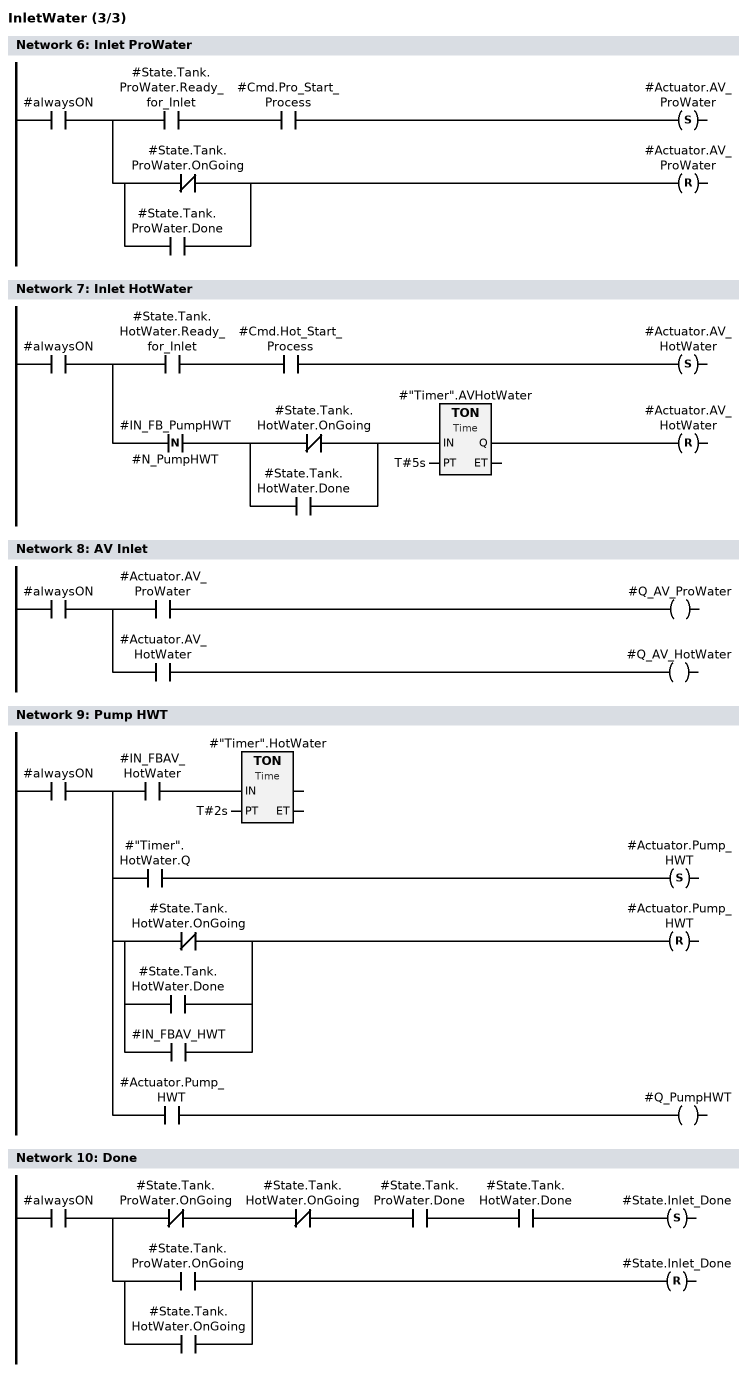
   RUNG wire#powerrail
      Contact( #alwaysON )
      wire#w1
      Contact( #State.Tank.ProWater.Ready_for_Inlet )
      Contact( #Cmd.Pro_Start_Process )
      S_Coil( #Actuator.AV_ProWater )
   END_RUNG
   RUNG wire#w1
      I_Contact( #State.Tank.ProWater.OnGoing )
      wire#w2
      R_Coil( #Actuator.AV_ProWater )
   END_RUNG
   RUNG wire#w1
      Contact( #State.Tank.ProWater.Done )
   END_RUNG wire#w2
   // the same network as SCL:
   IF #alwaysON AND #State.Tank.ProWater.Ready_for_Inlet AND #Cmd.Pro_Start_Process THEN
       #Actuator.AV_ProWater := TRUE;
   END_IF;
   IF #alwaysON AND (NOT #State.Tank.ProWater.OnGoing OR #State.Tank.ProWater.Done) THEN
       #Actuator.AV_ProWater := FALSE;
   END_IF;
END_REGION

REGION Network 7: Inlet HotWater
   RUNG wire#powerrail
      Contact( #alwaysON )
      wire#w1
      Contact( #State.Tank.HotWater.Ready_for_Inlet )
      Contact( #Cmd.Hot_Start_Process )
      S_Coil( #Actuator.AV_HotWater )
   END_RUNG
   RUNG wire#w1
      N_Contact(operand := #IN_FB_PumpHWT, bit := #N_PumpHWT)
      wire#w2
      I_Contact( #State.Tank.HotWater.OnGoing )
      wire#w3
      { S7_Templates := "time_type := Time" } #"Timer".AVHotWater.TON(pt := T#5s, et =>)
      R_Coil( #Actuator.AV_HotWater )
   END_RUNG
   RUNG wire#w2
      Contact( #State.Tank.HotWater.Done )
   END_RUNG wire#w3
   // the same network as SCL:
   IF #alwaysON AND #State.Tank.HotWater.Ready_for_Inlet AND #Cmd.Hot_Start_Process THEN
       #Actuator.AV_HotWater := TRUE;
   END_IF;
   #_w1 := #alwaysON AND NOT #IN_FB_PumpHWT AND #N_PumpHWT;   // falling edge of #IN_FB_PumpHWT
   #N_PumpHWT := #IN_FB_PumpHWT;
   #"Timer".AVHotWater.TON(IN := #_w1 AND (NOT #State.Tank.HotWater.OnGoing OR #State.Tank.HotWater.Done),
                           PT := T#5s);
   IF #"Timer".AVHotWater.Q THEN #Actuator.AV_HotWater := FALSE; END_IF;
END_REGION

REGION Network 8: AV Inlet
   RUNG wire#powerrail
      Contact( #alwaysON )
      wire#w1
      Contact( #Actuator.AV_ProWater )
      Coil( #Q_AV_ProWater )
   END_RUNG
   RUNG wire#w1
      Contact( #Actuator.AV_HotWater )
      Coil( #Q_AV_HotWater )
   END_RUNG
   // the same network as SCL:
   #Q_AV_ProWater := #alwaysON AND #Actuator.AV_ProWater;
   #Q_AV_HotWater := #alwaysON AND #Actuator.AV_HotWater;
END_REGION

REGION Network 9: Pump HWT
   RUNG wire#powerrail
      Contact( #alwaysON )
      wire#w1
      Contact( #IN_FBAV_HotWater )
      { S7_Templates := "time_type := Time" } #"Timer".HotWater.TON(pt := T#2s, et =>)
   END_RUNG
   RUNG wire#w1
      Contact( #"Timer".HotWater.Q )
      S_Coil( #Actuator.Pump_HWT )
   END_RUNG
   RUNG wire#w1
      I_Contact( #State.Tank.HotWater.OnGoing )
      wire#w2
      R_Coil( #Actuator.Pump_HWT )
   END_RUNG
   RUNG wire#w1
      Contact( #State.Tank.HotWater.Done )
   END_RUNG wire#w2
   RUNG wire#w1
      Contact( #IN_FBAV_HWT )
   END_RUNG wire#w2
   RUNG wire#w1
      Contact( #Actuator.Pump_HWT )
      Coil( #Q_PumpHWT )
   END_RUNG
   // the same network as SCL:
   #"Timer".HotWater.TON(IN := #alwaysON AND #IN_FBAV_HotWater, PT := T#2s);
   IF #alwaysON AND #"Timer".HotWater.Q THEN #Actuator.Pump_HWT := TRUE; END_IF;
   IF #alwaysON AND (NOT #State.Tank.HotWater.OnGoing OR #State.Tank.HotWater.Done OR #IN_FBAV_HWT) THEN
       #Actuator.Pump_HWT := FALSE;
   END_IF;
   #Q_PumpHWT := #alwaysON AND #Actuator.Pump_HWT;
END_REGION

REGION Network 10: Done
   RUNG wire#powerrail
      Contact( #alwaysON )
      wire#w1
      I_Contact( #State.Tank.ProWater.OnGoing )
      I_Contact( #State.Tank.HotWater.OnGoing )
      Contact( #State.Tank.ProWater.Done )
      Contact( #State.Tank.HotWater.Done )
      S_Coil( #State.Inlet_Done )
   END_RUNG
   RUNG wire#w1
      Contact( #State.Tank.ProWater.OnGoing )
      wire#w2
      R_Coil( #State.Inlet_Done )
   END_RUNG
   RUNG wire#w1
      Contact( #State.Tank.HotWater.OnGoing )
   END_RUNG wire#w2
   // the same network as SCL:
   IF #alwaysON AND NOT #State.Tank.ProWater.OnGoing AND NOT #State.Tank.HotWater.OnGoing AND #State.Tank.ProWater.Done AND #State.Tank.HotWater.Done THEN
       #State.Inlet_Done := TRUE;
   END_IF;
   IF #alwaysON AND (#State.Tank.ProWater.OnGoing OR #State.Tank.HotWater.OnGoing) THEN
       #State.Inlet_Done := FALSE;
   END_IF;
END_REGION
END_FUNCTION_BLOCK

FUNCTION_BLOCK "Storage Tank"   // FB7, LAD
{ S7_Optimized_Access := 'TRUE' }
VERSION : 0.1
// stored: AutoNumber true, IsIECCheckEnabled false, IsRetainMemResEnabled false, MemoryReserve 100, SetENOAutomatically false, UDAEnableTagReadback false
   VAR_INPUT
      Lock : Bool;
      Reset : Bool;
   END_VAR
   VAR_OUTPUT
      AV_Inlet : Bool;
   END_VAR
   VAR_IN_OUT
      Tank_Level : Real;
   END_VAR
   VAR
      Parameter : Struct
         Level_High : Real := 100.0;
         Level_Med : Real := 50.0;
         Level_Low : Real;
      END_STRUCT;
      State : Struct
         Tank_HL : Bool;
         Tank_ML : Bool;
         Tank_LL : Bool;
      END_STRUCT;
      Actuator : Struct
         AV_Inlet : Bool;
      END_STRUCT;
      AlwaysOn : Bool;
      Stat_Ready_for_Transfer : Bool;
      Ready_for_Transfer : Bool;
   END_VAR
BEGIN

REGION Network 1: Always On
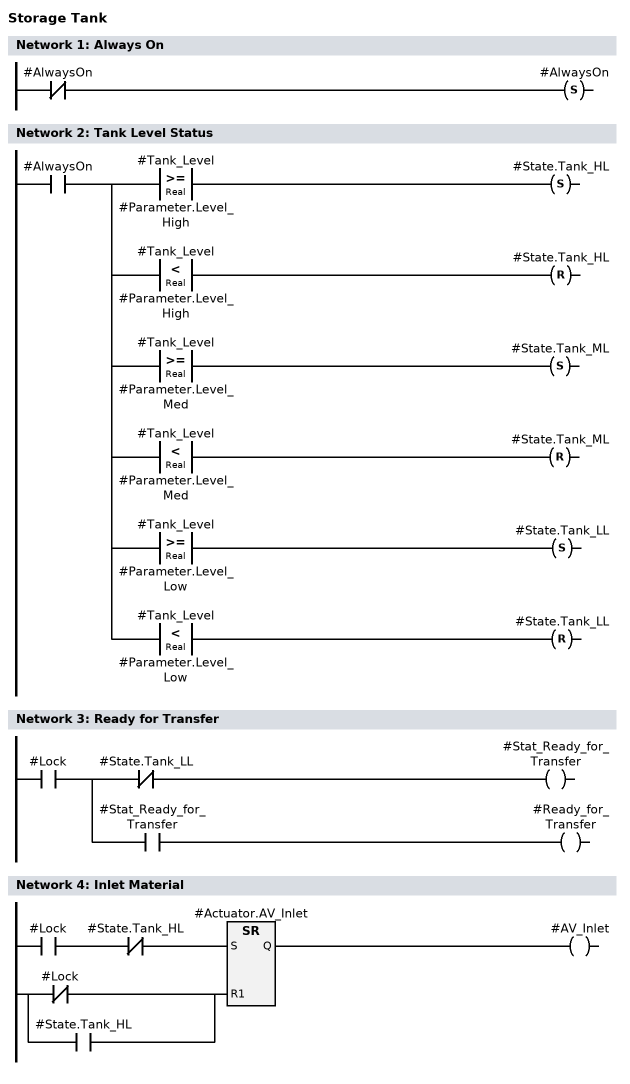
   RUNG wire#powerrail
      I_Contact( #AlwaysOn )
      S_Coil( #AlwaysOn )
   END_RUNG
   // the same network as SCL:
   IF NOT #AlwaysOn THEN #AlwaysOn := TRUE; END_IF;
END_REGION

REGION Network 2: Tank Level Status
   RUNG wire#powerrail
      Contact( #AlwaysOn )
      wire#w1
      { S7_Templates := "SrcType := Real" } GE_Contact(in1 := #Tank_Level, in2 := #Parameter.Level_High)
      S_Coil( #State.Tank_HL )
   END_RUNG
   RUNG wire#w1
      { S7_Templates := "SrcType := Real" } LT_Contact(in1 := #Tank_Level, in2 := #Parameter.Level_High)
      R_Coil( #State.Tank_HL )
   END_RUNG
   RUNG wire#w1
      { S7_Templates := "SrcType := Real" } GE_Contact(in1 := #Tank_Level, in2 := #Parameter.Level_Med)
      S_Coil( #State.Tank_ML )
   END_RUNG
   RUNG wire#w1
      { S7_Templates := "SrcType := Real" } LT_Contact(in1 := #Tank_Level, in2 := #Parameter.Level_Med)
      R_Coil( #State.Tank_ML )
   END_RUNG
   RUNG wire#w1
      { S7_Templates := "SrcType := Real" } GE_Contact(in1 := #Tank_Level, in2 := #Parameter.Level_Low)
      S_Coil( #State.Tank_LL )
   END_RUNG
   RUNG wire#w1
      { S7_Templates := "SrcType := Real" } LT_Contact(in1 := #Tank_Level, in2 := #Parameter.Level_Low)
      R_Coil( #State.Tank_LL )
   END_RUNG
   // the same network as SCL:
   IF #AlwaysOn AND (#Tank_Level >= #Parameter.Level_High) THEN #State.Tank_HL := TRUE; END_IF;
   IF #AlwaysOn AND (#Tank_Level < #Parameter.Level_High) THEN #State.Tank_HL := FALSE; END_IF;
   IF #AlwaysOn AND (#Tank_Level >= #Parameter.Level_Med) THEN #State.Tank_ML := TRUE; END_IF;
   IF #AlwaysOn AND (#Tank_Level < #Parameter.Level_Med) THEN #State.Tank_ML := FALSE; END_IF;
   IF #AlwaysOn AND (#Tank_Level >= #Parameter.Level_Low) THEN #State.Tank_LL := TRUE; END_IF;
   IF #AlwaysOn AND (#Tank_Level < #Parameter.Level_Low) THEN #State.Tank_LL := FALSE; END_IF;
END_REGION

REGION Network 3: Ready for Transfer
   RUNG wire#powerrail
      Contact( #Lock )
      wire#w1
      I_Contact( #State.Tank_LL )
      Coil( #Stat_Ready_for_Transfer )
   END_RUNG
   RUNG wire#w1
      Contact( #Stat_Ready_for_Transfer )
      Coil( #Ready_for_Transfer )
   END_RUNG
   // the same network as SCL:
   #Stat_Ready_for_Transfer := #Lock AND NOT #State.Tank_LL;
   #Ready_for_Transfer := #Lock AND #Stat_Ready_for_Transfer;
END_REGION

REGION Network 4: Inlet Material
   RUNG wire#powerrail
      Contact( #Lock )
      I_Contact( #State.Tank_HL )
      S_SR(operand := #Actuator.AV_Inlet, r1 := wire#w1)
      Coil( #AV_Inlet )
   END_RUNG
   RUNG wire#powerrail
      I_Contact( #Lock )
   END_RUNG wire#w1
   RUNG wire#powerrail
      Contact( #State.Tank_HL )
   END_RUNG wire#w1
   // the same network as SCL:
   IF #Lock AND NOT #State.Tank_HL THEN
       #Actuator.AV_Inlet := TRUE;   // SR flip-flop
   END_IF;
   IF NOT #Lock OR #State.Tank_HL THEN #Actuator.AV_Inlet := FALSE; END_IF;
   #AV_Inlet := #Actuator.AV_Inlet;
END_REGION
END_FUNCTION_BLOCK

FUNCTION "IO Blending" : Void   // FC3, LAD
{ S7_Optimized_Access := 'TRUE' }
VERSION : 0.1
// stored: AutoNumber true, IsIECCheckEnabled false, SetENOAutomatically false, UDAEnableTagReadback false
BEGIN
END_FUNCTION

FUNCTION_BLOCK "IO_Valve_Blending"   // FB2, LAD
{ S7_Optimized_Access := 'FALSE' }
VERSION : 0.1
// stored: AutoNumber true, IsIECCheckEnabled false, SetENOAutomatically false, UDAEnableTagReadback false
   VAR_INPUT
      lock : Bool;
      Init : Bool;
      Reset : Bool;
   END_VAR
   VAR
      "AV-20.01" { S7_SetPoint := 'True'} : "Valve";   // AUTO BUTTERFLY VALVE OUTLET PRODUCT BLENDING TANK T-20.00
      "AV-20.02" { S7_SetPoint := 'True'} : "Valve";   // AUTO BUTTERGLY VALVE INLET CIP SUPPLY LINE BLENDING TANK T-20.00
      "AV-20.03" { S7_SetPoint := 'True'} : "Valve";   // AUTO BUTTERFLY VALVE OUTLET PRODUCT FROM BLENDING T-20.00 TO TRANSFER PUMP P-21.01
      "AV-20.04" { S7_SetPoint := 'True'} : "Valve";   // AUTO BUTTERFLY VALVE CIP RETURN FROM BLENDING TANK T-20.00
      "AV-20.05" { S7_SetPoint := 'True'} : "Valve";   // AUTO BUTTERFLY VALVE INLET FRESH CHILI FROM T-06.00 TO BLENDING TANK T-20.00
      "AV-20.06" { S7_SetPoint := 'True'} : "Valve";   // AUTO BUTTERFLY VALVE INLET FRESH CHILI FROM T-07.00 TO BLENDING TANK T-20.00
      "AV-20.07" { S7_SetPoint := 'True'} : "Valve";   // AUTO BUTTERFLY VALVE INLET FRESH CHILI FROM T-08.00 TO BLENDING TANK T-20.00
      "AV-20.08" { S7_SetPoint := 'True'} : "Valve";   // AUTO BUTTERFLY VALVE INLET GARLIC FROM T-09.00 TO BLENDING TANK T-20.00
      "AV-20.09" { S7_SetPoint := 'True'} : "Valve";   // AUTO BUTTERFLY VALVE INLET CHILI AWETAN FROM T-02.00 TO BLENDING TANK T-20.00
      "AV-20.10" { S7_SetPoint := 'True'} : "Valve";   // AUTO BUTTERFLY VALVE INLET CHILI AWETAN FROM T-03.00 TO BLENDING TANK T-20.00
      "AV-20.11" { S7_SetPoint := 'True'} : "Valve";   // AUTO BUTTERFLY VALVE INLET CHILI AWETAN FROM T-04.00 TO BLENDING TANK T-20.00
      "AV-20.12" { S7_SetPoint := 'True'} : "Valve";   // AUTO BUTTERFLY VALVE INLET TOMATO FROM T-05.00 TO BLENDING TANK T-20.00
      "AV-20.13" { S7_SetPoint := 'True'} : "Valve";   // AUTO BUTTERFLY VALVE INLET PRODUCT FROM REWORK T-22.00 TO BLENDING TANK T-20.00
      "AV-20.14" { S7_SetPoint := 'True'} : "Valve";   // AUTO BUTTERFLY VALVE INLET INGRIDIENT FROM HOMOMIXER T-12.00 TO BLENDING TANK T-20.00
      "AV-20.15" { S7_SetPoint := 'True'} : "Valve";   // AUTO BUTTERFLY VALVE INLET VINEGAR FROM T-10.00 TO BLENDING TANK T-20.00
      "AV-20.16" { S7_SetPoint := 'True'} : "Valve";   // AUTO BUTTERFLY VALVE INLET PROCESS WATER TO BLENDING TANK T-20.00
      "AV-20.17" { S7_SetPoint := 'True'} : "Valve";   // AUTO BUTTERFLY VALVE INLET SUGAR DISSOLVING TO BLENDING TANK T-20.00
      "AV-20.31" { S7_SetPoint := 'True'} : "Valve";   // AUTO BUTTERFLY VALVE INLET CIP SUPPLY SIDE 1 BLENDING TANK T-20.00
      "AV-20.32" { S7_SetPoint := 'True'} : "Valve";   // AUTO BUTTERFLY VALVE INLET CIP SUPPLY SIDE 2 BLENDING TANK T-20.00
      "AV-20.33" { S7_SetPoint := 'True'} : "Valve";   // AUTO BUTTERFLY VALVE INLET CIP SUPPLY TO BLENDING TANK T-20.00
      "AV-20.34" { S7_SetPoint := 'True'} : "Valve";   // AUTO BUTTERFLY VALVE INLET CIP SUPPLY TO PIPE LINE TOMATO BLENDING TANK T-20.00
      "AV-20.35" { S7_SetPoint := 'True'} : "Valve";   // AUTO BUTTERFLY VALVE INLET CIP SUPPLY TO PIPE LINE CHILI AWETAN 4 BLENDING TANK T-20.00
      "AV-20.36" { S7_SetPoint := 'True'} : "Valve";   // AUTO BUTTERFLY VALVE INLET CIP SUPPLY TO PIPE LINE CHILI AWETAN 3 BLENDING TANK T-20.00
      "AV-20.37" { S7_SetPoint := 'True'} : "Valve";   // AUTO BUTTERFLY VALVE INLET CIP SUPPLY TO PIPE LINE CHILI AWETAN 2 BLENDING TANK T-20.00
      "AV-20.38" { S7_SetPoint := 'True'} : "Valve";   // AUTO BUTTERFLY VALVE INLET CIP SUPPLY TO PIPE LINE GARLIC BLENDING TANK T-20.00
      "AV-20.39" { S7_SetPoint := 'True'} : "Valve";   // AUTO BUTTERFLY VALVE INLET CIP SUPPLY TO PIPE LINE FRESH CHILI 8 BLENDING TANK T-20.00
      "AV-20.40" { S7_SetPoint := 'True'} : "Valve";   // AUTO BUTTERFLY VALVE INLET CIP SUPPLY TO PIPE LINE FRESH CHILI 7 BLENDING TANK T-20.00
      "AV-20.41" { S7_SetPoint := 'True'} : "Valve";   // AUTO BUTTERFLY VALVE INLET CIP SUPPLY TO PIPE LINE FRESH CHILI 6 BLENDING TANK T-20.00
      "AV-21.01" { S7_SetPoint := 'True'} : "Valve";   // AUTO BUTTERFLY VALVE OUTLET PRODUCT BLENDING TANK T-21.00
      "AV-21.02" { S7_SetPoint := 'True'} : "Valve";   // AUTO BUTTERFLY VALVE INLET CIP SUPPLY LINE BLENDING TANK T-21.00
      "AV-21.03" { S7_SetPoint := 'True'} : "Valve";   // AUTO BUTTERFLY VALVE OUTLET PRODUCT FROM BLENDING T-21.00 TO TRANSFER PUMP P-21.01
      "AV-21.04" { S7_SetPoint := 'True'} : "Valve";   // AUTO BUTTERFLY VALVE CIP RETURN FROM BLENDING TANK T-21.00
      "AV-21.05" { S7_SetPoint := 'True'} : "Valve";   // AUTO BUTTERFLY VALVE INLET FRESH CHILI FROM T-06.00 TO BLENDING TANK T-21.00
      "AV-21.06" { S7_SetPoint := 'True'} : "Valve";   // AUTO BUTTERFLY VALVE INLET FRESH CHILI FROM T-07.00 TO BLENDING TANK T-21.00
      "AV-21.07" { S7_SetPoint := 'True'} : "Valve";   // AUTO BUTTERFLY VALVE INLET FRESH CHILI FROM T-08.00 TO BLENDING TANK T-21.00
      "AV-21.08" { S7_SetPoint := 'True'} : "Valve";   // AUTO BUTTERFLY VALVE INLET GARLIC FROM T-09.00 TO BLENDING TANK T-21.00
      "AV-21.09" { S7_SetPoint := 'True'} : "Valve";   // AUTO BUTTERFLY VALVE INLET CHILI AWETAN FROM T-02.00 TO BLENDING TANK T-21.00
      "AV-21.10" { S7_SetPoint := 'True'} : "Valve";   // AUTO BUTTERFLY VALVE INLET CHILI AWETAN FROM T-03.00 TO BLENDING TANK T-21.00
      "AV-21.11" { S7_SetPoint := 'True'} : "Valve";   // AUTO BUTTERFLY VALVE INLET CHILI AWETAN FROM T-04.00 TO BLENDING TANK T-21.00
      "AV-21.12" { S7_SetPoint := 'True'} : "Valve";   // AUTO BUTTERFLY VALVE INLET TOMATO FROM T-05.00 TO BLENDING TANK T-21.00
      "AV-21.13" { S7_SetPoint := 'True'} : "Valve";   // AUTO BUTTERFLY VALVE INLET PRODUCT FROM REWORK T-22.00 TO BLENDING TANK T-21.00
      "AV-21.14" { S7_SetPoint := 'True'} : "Valve";   // AUTO BUTTERFLY VALVE INLET INGRIDIENT FROM HOMOMIXER T-12.00 TO BLENDING TANK T-21.00
      "AV-21.15" { S7_SetPoint := 'True'} : "Valve";   // AUTO BUTTERFLY VALVE INLET VINEGAR FROM T-10.00 TO BLENDING TANK T-21.00
      "AV-21.16" { S7_SetPoint := 'True'} : "Valve";   // AUTO BUTTERFLY VALVE INLET PROCESS WATER TO BLENDING TANK T-21.00
      "AV-21.17" { S7_SetPoint := 'True'} : "Valve";   // AUTO BUTTERFLY VALVE INLET SUGAR DISSOLVING TO BLENDING TANK T-21.00
      "AV-21.18" { S7_SetPoint := 'True'} : "Valve";   // AUTO BUTTERFLY VALVE DRAIN REWORK TANK LINE THE-4
      "AV-21.31" { S7_SetPoint := 'True'} : "Valve";   // AUTO BUTTERFLY VALVE INLET CIP SUPPLY SIDE 1 BLENDING TANK T-21.00
      "AV-21.32" { S7_SetPoint := 'True'} : "Valve";   // AUTO BUTTERFLY VALVE INLET CIP SUPPLY SIDE 2 BLENDING TANK T-21.00
      "AV-21.33" { S7_SetPoint := 'True'} : "Valve";   // AUTO BUTTERFLY VALVE INLET CIP SUPPLY TO BLENDING TANK T-21.00
      "AV-21.34" { S7_SetPoint := 'True'} : "Valve";   // AUTO BUTTERFLY VALVE INLET CIP SUPPLY TO PIPE LINE TOMATO BLENDING TANK T-21.00
      "AV-21.35" { S7_SetPoint := 'True'} : "Valve";   // AUTO BUTTERFLY VALVE INLET CIP SUPPLY TO PIPE LINE CHILI AWETAN 4 BLENDING TANK T-21.00
      "AV-21.36" { S7_SetPoint := 'True'} : "Valve";   // AUTO BUTTERFLY VALVE INLET CIP SUPPLY TO PIPE LINE CHILI AWETAN 3 BLENDING TANK T-21.00
      "AV-21.37" { S7_SetPoint := 'True'} : "Valve";   // AUTO BUTTERFLY VALVE INLET CIP SUPPLY TO PIPE LINE CHILI AWETAN 2 BLENDING TANK T-21.00
      "AV-21.38" { S7_SetPoint := 'True'} : "Valve";   // AUTO BUTTERFLY VALVE INLET CIP SUPPLY TO PIPE LINE GARLIC BLENDING TANK T-21.00
      "AV-21.39" { S7_SetPoint := 'True'} : "Valve";   // AUTO BUTTERFLY VALVE INLET CIP SUPPLY TO PIPE LINE FRESH CHILI 8 BLENDING TANK T-21.00
      "AV-21.40" { S7_SetPoint := 'True'} : "Valve";   // AUTO BUTTERFLY VALVE INLET CIP SUPPLY TO PIPE LINE FRESH CHILI 7 BLENDING TANK T-21.00
      "AV-21.41" { S7_SetPoint := 'True'} : "Valve";   // AUTO BUTTERFLY VALVE INLET CIP SUPPLY TO PIPE LINE FRESH CHILI 6 BLENDING TANK T-21.00
      "AV-22.01" { S7_SetPoint := 'True'} : "Valve";   // AUTO BUTTERFLY VALVE OUTLET PRODUCT FROM REWORK T-22.00 TO TRANSFER PUMP P-22.01
      "AV-22.02" { S7_SetPoint := 'True'} : "Valve";   // AUTO BUTTERFLY VALVE CIP SUPPLY FROM REWORK & LINE TO CIP SUPPLY PUMP P-22.02
      "AV-22.03" { S7_SetPoint := 'True'} : "Valve";   // AUTO BUTTERFLY VALVE DRAIN MONO PUMP P-22.01
      "AV-22.06" { S7_SetPoint := 'True'} : "Valve";   // AUTO BUTTERFLY VALVE CIP SUPPLY REWORK TANK T-22.00
      "AV-22.11" { S7_SetPoint := 'True'} : "Valve";   // AUTO BUTTERFLY VALVE MAIN CIP SUPPLY BLENDING TANKS THE-4
      "AV-22.21" { S7_SetPoint := 'True'} : "Valve";   // AUTO BUTTERFLY VALVE CIP RETURN BLENDING TANK THE-4 LINE 1
      "AV-22.22" { S7_SetPoint := 'True'} : "Valve";   // AUTO BUTTERFLY VALVE CIP RETURN BLENDING TANK THE-4 LINE 2
      "AV-30.01" { S7_SetPoint := 'True'} : "Valve";   // AUTO BUTTERFLY VALVE OUTLET PRODUCT BLENDING TANK T-30.00
      "AV-30.02" { S7_SetPoint := 'True'} : "Valve";   // AUTO BUTTERFLY VALVE INLET CIP SUPPLY LINE BLENDING TANK T-30.00
      "AV-30.03" { S7_SetPoint := 'True'} : "Valve";   // AUTO BUTTERFLY VALVE OUTLET PRODUCT FROM BLENDING T-30.00 TO TRANSFER PUMP P-31.01
      "AV-30.04" { S7_SetPoint := 'True'} : "Valve";   // AUTO BUTTERFLY VALVE CIP RETURN FROM BLENDING TANK T-30.00
      "AV-30.05" { S7_SetPoint := 'True'} : "Valve";   // AUTO BUTTERFLY VALVE INLET FRESH CHILI FROM T-06.00 TO BLENDING TANK T-30.00
      "AV-30.06" { S7_SetPoint := 'True'} : "Valve";   // AUTO BUTTERFLY VALVE INLET FRESH CHILI FROM T-07.00 TO BLENDING TANK T-30.00
      "AV-30.07" { S7_SetPoint := 'True'} : "Valve";   // AUTO BUTTERFLY VALVE INLET FRESH CHILI FROM T-08.00 TO BLENDING TANK T-30.00
      "AV-30.08" { S7_SetPoint := 'True'} : "Valve";   // AUTO BUTTERFLY VALVE INLET GARLIC FROM T-09.00 TO BLENDING TANK T-30.00
      "AV-30.09" { S7_SetPoint := 'True'} : "Valve";   // AUTO BUTTERFLY VALVE INLET CHILI AWETAN FROM T-02.00 TO BLENDING TANK T-30.00
      "AV-30.10" { S7_SetPoint := 'True'} : "Valve";   // AUTO BUTTERFLY VALVE INLET CHILI AWETAN FROM T-03.00 TO BLENDING TANK T-30.00
      "AV-30.11" { S7_SetPoint := 'True'} : "Valve";   // AUTO BUTTERFLY VALVE INLET CHILI AWETAN FROM T-04.00 TO BLENDING TANK T-30.00
      "AV-30.12" { S7_SetPoint := 'True'} : "Valve";   // AUTO BUTTERFLY VALVE INLET TOMATO FROM T-05.00 TO BLENDING TANK T-30.00
      "AV-30.13" { S7_SetPoint := 'True'} : "Valve";   // AUTO BUTTERFLY VALVE INLET PRODUCT FROM REWORK T-22.00 TO BLENDING TANK T-30.00
      "AV-30.14" { S7_SetPoint := 'True'} : "Valve";   // AUTO BUTTERFLY VALVE INLET INGRIDIENT FROM HOMOMIXER T-12.00 TO BLENDING TANK T-30.00
      "AV-30.15" { S7_SetPoint := 'True'} : "Valve";   // AUTO BUTTERFLY VALVE INLET VINEGAR FROM T-10.00 TO BLENDING TANK T-30.00
      "AV-30.16" { S7_SetPoint := 'True'} : "Valve";   // AUTO BUTTERFLY VALVE INLET PROCESS WATER TO BLENDING TANK T-30.00
      "AV-30.17" { S7_SetPoint := 'True'} : "Valve";   // AUTO BUTTERFLY VALVE INLET SUGAR DISSOLVING TO BLENDING TANK T-30.00
      "AV-30.31" { S7_SetPoint := 'True'} : "Valve";   // AUTO BUTTERFLY VALVE INLET CIP SUPPLY SIDE 1 BLENDING TANK T-30.00
      "AV-30.32" { S7_SetPoint := 'True'} : "Valve";   // AUTO BUTTERFLY VALVE INLET CIP SUPPLY SIDE 2 BLENDING TANK T-30.00
      "AV-30.33" { S7_SetPoint := 'True'} : "Valve";   // AUTO BUTTERFLY VALVE INLET CIP SUPPLY TO BLENDING TANK T-30.00
      "AV-30.34" { S7_SetPoint := 'True'} : "Valve";   // AUTO BUTTERFLY VALVE INLET CIP SUPPLY TO PIPE LINE TOMATO BLENDING TANK T-30.00
      "AV-30.35" { S7_SetPoint := 'True'} : "Valve";   // AUTO BUTTERFLY VALVE INLET CIP SUPPLY TO PIPE LINE CHILI AWETAN 4 BLENDING TANK T-30.00
      "AV-30.36" { S7_SetPoint := 'True'} : "Valve";   // AUTO BUTTERFLY VALVE INLET CIP SUPPLY TO PIPE LINE CHILI AWETAN 3 BLENDING TANK T-30.00
      "AV-30.37" { S7_SetPoint := 'True'} : "Valve";   // AUTO BUTTERFLY VALVE INLET CIP SUPPLY TO PIPE LINE CHILI AWETAN 2 BLENDING TANK T-30.00
      "AV-30.38" { S7_SetPoint := 'True'} : "Valve";   // AUTO BUTTERFLY VALVE INLET CIP SUPPLY TO PIPE LINE GARLIC BLENDING TANK T-30.00
      "AV-30.39" { S7_SetPoint := 'True'} : "Valve";   // AUTO BUTTERFLY VALVE INLET CIP SUPPLY TO PIPE LINE FRESH CHILI 8 BLENDING TANK T-30.00
      "AV-30.40" { S7_SetPoint := 'True'} : "Valve";   // AUTO BUTTERFLY VALVE INLET CIP SUPPLY TO PIPE LINE FRESH CHILI 7 BLENDING TANK T-30.00
      "AV-30.41" { S7_SetPoint := 'True'} : "Valve";   // AUTO BUTTERFLY VALVE INLET CIP SUPPLY TO PIPE LINE FRESH CHILI 6 BLENDING TANK T-30.00
      "AV-31.01" { S7_SetPoint := 'True'} : "Valve";   // AUTO BUTTERFLY VALVE OUTLET PRODUCT BLENDING TANK T-31.00
      "AV-31.02" { S7_SetPoint := 'True'} : "Valve";   // AUTO BUTTERFLY VALVE INLET CIP SUPPLY LINE BLENDING TANK T-31.00
      "AV-31.03" { S7_SetPoint := 'True'} : "Valve";   // AUTO BUTTERFLY VALVE OUTLET PRODUCT FROM BLENDING T-31.00 TO TRANSFER PUMP P-31.01
      "AV-31.04" { S7_SetPoint := 'True'} : "Valve";   // AUTO BUTTERFLY VALVE CIP RETURN FROM BLENDING TANK T-31.00
      "AV-31.05" { S7_SetPoint := 'True'} : "Valve";   // AUTO BUTTERFLY VALVE INLET FRESH CHILI FROM T-06.00 TO BLENDING TANK T-31.00
      "AV-31.06" { S7_SetPoint := 'True'} : "Valve";   // AUTO BUTTERFLY VALVE INLET FRESH CHILI FROM T-07.00 TO BLENDING TANK T-31.00
      "AV-31.07" { S7_SetPoint := 'True'} : "Valve";   // AUTO BUTTERFLY VALVE INLET FRESH CHILI FROM T-08.00 TO BLENDING TANK T-31.00
      "AV-31.08" { S7_SetPoint := 'True'} : "Valve";   // AUTO BUTTERFLY VALVE INLET GARLIC FROM T-09.00 TO BLENDING TANK T-31.00
      "AV-31.09" { S7_SetPoint := 'True'} : "Valve";   // AUTO BUTTERFLY VALVE INLET CHILI AWETAN FROM T-02.00 TO BLENDING TANK T-31.00
      "AV-31.10" { S7_SetPoint := 'True'} : "Valve";   // AUTO BUTTERFLY VALVE INLET CHILI AWETAN FROM T-03.00 TO BLENDING TANK T-31.00
      "AV-31.11" { S7_SetPoint := 'True'} : "Valve";   // AUTO BUTTERFLY VALVE INLET CHILI AWETAN FROM T-04.00 TO BLENDING TANK T-31.00
      "AV-31.12" { S7_SetPoint := 'True'} : "Valve";   // AUTO BUTTERFLY VALVE INLET TOMATO FROM T-05.00 TO BLENDING TANK T-31.00
      "AV-31.13" { S7_SetPoint := 'True'} : "Valve";   // AUTO BUTTERFLY VALVE INLET PRODUCT FROM REWORK T-22.00 TO BLENDING TANK T-31.00
      "AV-31.14" { S7_SetPoint := 'True'} : "Valve";   // AUTO BUTTERFLY VALVE INLET INGRIDIENT FROM HOMOMIXER T-12.00 TO BLENDING TANK T-31.00
      "AV-31.15" { S7_SetPoint := 'True'} : "Valve";   // AUTO BUTTERFLY VALVE INLET VINEGAR FROM T-10.00 TO BLENDING TANK T-31.00
      "AV-31.16" { S7_SetPoint := 'True'} : "Valve";   // AUTO BUTTERFLY VALVE INLET PROCESS WATER TO BLENDING TANK T-31.00
      "AV-31.17" { S7_SetPoint := 'True'} : "Valve";   // AUTO BUTTERFLY VALVE INLET SUGAR DISSOLVING TO BLENDING TANK T-31.00
      "AV-31.18" { S7_SetPoint := 'True'} : "Valve";   // AUTO BUTTERFLY VALVE DRAIN REWORK TANK LINE THE-5
      "AV-31.31" { S7_SetPoint := 'True'} : "Valve";   // AUTO BUTTERFLY VALVE INLET CIP SUPPLY SIDE 1 BLENDING TANK T-31.00
      "AV-31.32" { S7_SetPoint := 'True'} : "Valve";   // AUTO BUTTERFLY VALVE INLET CIP SUPPLY SIDE 2 BLENDING TANK T-31.00
      "AV-31.33" { S7_SetPoint := 'True'} : "Valve";   // AUTO BUTTERFLY VALVE INLET CIP SUPPLY TO BLENDING TANK T-31.00
      "AV-31.34" { S7_SetPoint := 'True'} : "Valve";   // AUTO BUTTERFLY VALVE INLET CIP SUPPLY TO PIPE LINE TOMATO BLENDING TANK T-31.00
      "AV-31.35" { S7_SetPoint := 'True'} : "Valve";   // AUTO BUTTERFLY VALVE INLET CIP SUPPLY TO PIPE LINE CHILI AWETAN 4 BLENDING TANK T-31.00
      "AV-31.36" { S7_SetPoint := 'True'} : "Valve";   // AUTO BUTTERFLY VALVE INLET CIP SUPPLY TO PIPE LINE CHILI AWETAN 3 BLENDING TANK T-31.00
      "AV-31.37" { S7_SetPoint := 'True'} : "Valve";   // AUTO BUTTERFLY VALVE INLET CIP SUPPLY TO PIPE LINE CHILI AWETAN 2 BLENDING TANK T-31.00
      "AV-31.38" { S7_SetPoint := 'True'} : "Valve";   // AUTO BUTTERFLY VALVE INLET CIP SUPPLY TO PIPE LINE GARLIC BLENDING TANK T-31.00
      "AV-31.39" { S7_SetPoint := 'True'} : "Valve";   // AUTO BUTTERFLY VALVE INLET CIP SUPPLY TO PIPE LINE FRESH CHILI 8 BLENDING TANK T-31.00
      "AV-31.40" { S7_SetPoint := 'True'} : "Valve";   // AUTO BUTTERFLY VALVE INLET CIP SUPPLY TO PIPE LINE FRESH CHILI 7 BLENDING TANK T-31.00
      "AV-31.41" { S7_SetPoint := 'True'} : "Valve";   // AUTO BUTTERFLY VALVE INLET CIP SUPPLY TO PIPE LINE FRESH CHILI 6 BLENDING TANK T-31.00
      "AV-31.51" { S7_SetPoint := 'True'} : "Valve";   // AUTO BUTTERFLY VALVE DRAIN LINE TOMATO T-05.00
      "AV-31.52" { S7_SetPoint := 'True'} : "Valve";   // AUTO BUTTERFLY VALVE DRAIN LINE FRESH CHILI T-06.00
      "AV-31.53" { S7_SetPoint := 'True'} : "Valve";   // AUTO BUTTERFLY VALVE DRAIN LINE FRESH CHILI T-07.00
      "AV-31.54" { S7_SetPoint := 'True'} : "Valve";   // AUTO BUTTERFLY VALVE DRAIN LINE FRESH CHILI T-08.00
      "AV-31.55" { S7_SetPoint := 'True'} : "Valve";   // AUTO BUTTERFLY VALVE DRAIN LINE CHILI AWETAN T-02.00
      "AV-31.56" { S7_SetPoint := 'True'} : "Valve";   // AUTO BUTTERFLY VALVE DRAIN LINE CHILI AWETAN T-03.00 VALVE CLOSE POSITION
      "AV-31.57" { S7_SetPoint := 'True'} : "Valve";   // AUTO BUTTERFLY VALVE DRAIN LINE CHILI AWETAN T-04.00 VALVE CLOSE POSITION
      "AV-31.58" { S7_SetPoint := 'True'} : "Valve";   // AUTO BUTTERFLY VALVE DRAIN LINE GARLIC T-09.00 VALVE CLOSE POSITION
      "AV-31.59" { S7_SetPoint := 'True'} : "Valve";   // AUTO BUTTERFLY VALVE DRAIN LINE VINEGAR T-10.00 VALVE CLOSE POSITION
      "AV-31.60" { S7_SetPoint := 'True'} : "Valve";   // AUTO BUTTERFLY VALVE DRAIN LINE SUGAR DISSOLVING T-15.00 VALVE CLOSE POSITION
      "AV-31.61" { S7_SetPoint := 'True'} : "Valve";   // AUTO BUTTERFLY VALVE DRAIN LINES
      "AV-31.62" { S7_SetPoint := 'True'} : "Valve";   // AUTO BUTTERFLY VALVE CIP RETURN LINE 1
      "AV-32.01" { S7_SetPoint := 'True'} : "Valve";   // AUTO BUTTERFLY VALVE OUTLET PRODUCT FROM REWORK T-32.00 TO TRANSFER PUMP P-32.01
      "AV-32.02" { S7_SetPoint := 'True'} : "Valve";   // AUTO BUTTERFLY VALVE CIP SUPPLY FROM REWORK & LINE TO CIP SUPPLY PUMP P-32.02
      "AV-32.03" { S7_SetPoint := 'True'} : "Valve";   // AUTO BUTTERFLY VALVE DRAIN MONO PUMP P-32.01
      "AV-32.06" { S7_SetPoint := 'True'} : "Valve";   // AUTO BUTTERFLY VALVE CIP SUPPLY REWORK TANK T-32.00
      "AV-32.11" { S7_SetPoint := 'True'} : "Valve";   // AUTO BUTTERFLY VALVE MAIN CIP SUPPLY BLENDING TANKS THE-5
      "AV-32.21" { S7_SetPoint := 'True'} : "Valve";   // AUTO BUTTERFLY VALVE CIP RETURN BLENDING TANK THE-5 LINE 1
      "AV-32.22" { S7_SetPoint := 'True'} : "Valve";   // AUTO BUTTERFLY VALVE CIP RETURN BLENDING TANK THE-5 LINE 2
      "AV-20.42" { S7_SetPoint := 'True'} : "Valve";   // AUTO BUTTERFLY VALVE MAIN CIP SUPPLY BLENDING TANK T-20.00
      "AV-21.42" { S7_SetPoint := 'True'} : "Valve";   // AUTO BUTTERFLY VALVE MAIN CIP SUPPLY BLENDING TANK T-21.00
      "AV-22.04" { S7_SetPoint := 'True'} : "Valve";   // AUTO BUTTERFLY VALVE MAIN CIP SUPPLY REWORK TANK T-22.00
      "AV-22.05" { S7_SetPoint := 'True'} : "Valve";   // AUTO BUTTERFLY VALVE MAIN CIP SUPPLY LINE BLENDING TANK THE-4
      "AV-30.42" { S7_SetPoint := 'True'} : "Valve";   // AUTO BUTTERFLY VALVE MAIN CIP SUPPLY BLENDING TANK T-30.00
      "AV-31.42" { S7_SetPoint := 'True'} : "Valve";   // AUTO BUTTERFLY VALVE MAIN CIP SUPPLY BLENDING TANK T-31.00
      "AV-32.04" { S7_SetPoint := 'True'} : "Valve";   // AUTO BUTTERFLY VALVE MAIN CIP SUPPLY REWORK TANK T-32.00
      "AV-32.05" { S7_SetPoint := 'True'} : "Valve";   // AUTO BUTTERFLY VALVE MAIN CIP SUPPLY LINE BLENDING TANK THE-5
   END_VAR
   // "AV-20.05".OPdwCmd := 16#0008_0000;
BEGIN

REGION Network 1: AV-20.01
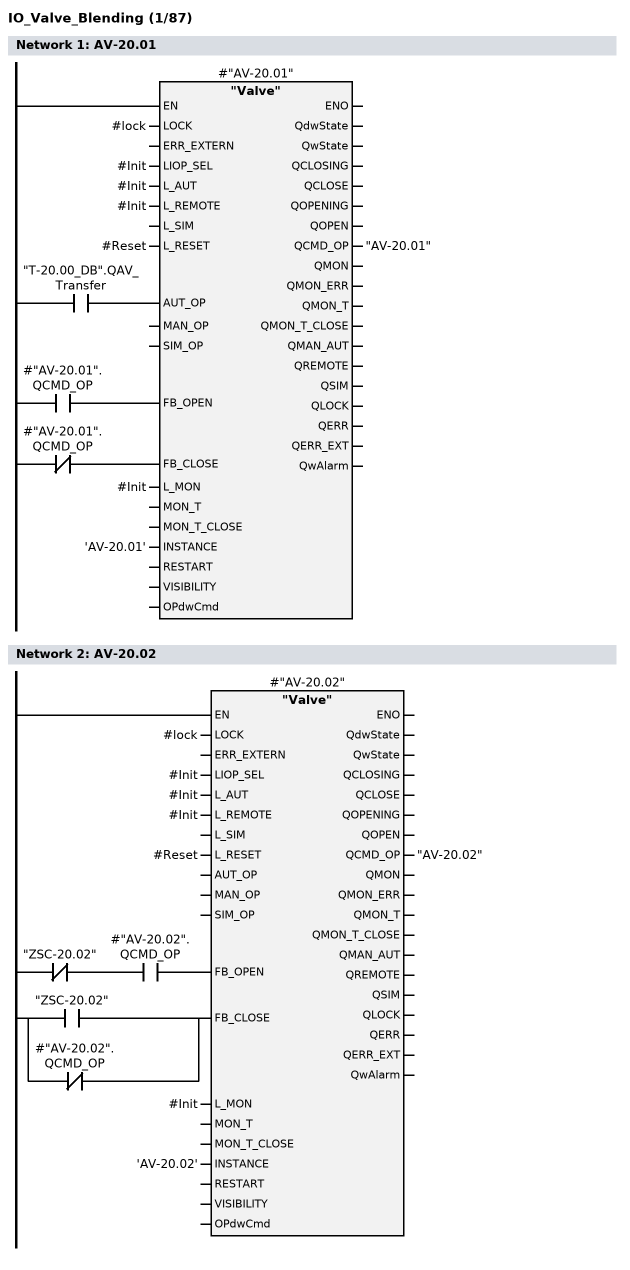
   RUNG wire#powerrail
      #"AV-20.01"(AUT_OP := wire#w1, FB_OPEN := wire#w2, FB_CLOSE := wire#w3, LOCK := #lock, ERR_EXTERN :=, LIOP_SEL := #Init, L_AUT := #Init, L_REMOTE := #Init, L_SIM :=, L_RESET := #Reset, MAN_OP :=, SIM_OP :=, L_MON := #Init, MON_T :=, MON_T_CLOSE :=, INSTANCE := 'AV-20.01', RESTART :=, VISIBILITY :=, OPdwCmd :=, QdwState =>, QwState =>, QCLOSING =>, QCLOSE =>, QOPENING =>, QOPEN =>, QCMD_OP => "AV-20.01", QMON =>, QMON_ERR =>, QMON_T =>, QMON_T_CLOSE =>, QMAN_AUT =>, QREMOTE =>, QSIM =>, QLOCK =>, QERR =>, QERR_EXT =>, QwAlarm =>)
   END_RUNG
   RUNG wire#powerrail
      Contact( "T-20.00_DB".QAV_Transfer )
   END_RUNG wire#w1
   RUNG wire#powerrail
      Contact( #"AV-20.01".QCMD_OP )
   END_RUNG wire#w2
   RUNG wire#powerrail
      I_Contact( #"AV-20.01".QCMD_OP )
   END_RUNG wire#w3
   // the same network as SCL:
   #"AV-20.01"(LOCK := #lock,   // "Valve"
               LIOP_SEL := #Init,
               L_AUT := #Init,
               L_REMOTE := #Init,
               L_RESET := #Reset,
               AUT_OP := "T-20.00_DB".QAV_Transfer,
               FB_OPEN := #"AV-20.01".QCMD_OP,
               FB_CLOSE := NOT #"AV-20.01".QCMD_OP,
               L_MON := #Init,
               INSTANCE := 'AV-20.01',
               QCMD_OP => "AV-20.01");
END_REGION

REGION Network 2: AV-20.02
   RUNG wire#powerrail
      #"AV-20.02"(FB_OPEN := wire#w1, FB_CLOSE := wire#w2, LOCK := #lock, ERR_EXTERN :=, LIOP_SEL := #Init, L_AUT := #Init, L_REMOTE := #Init, L_SIM :=, L_RESET := #Reset, AUT_OP :=, MAN_OP :=, SIM_OP :=, L_MON := #Init, MON_T :=, MON_T_CLOSE :=, INSTANCE := 'AV-20.02', RESTART :=, VISIBILITY :=, OPdwCmd :=, QdwState =>, QwState =>, QCLOSING =>, QCLOSE =>, QOPENING =>, QOPEN =>, QCMD_OP => "AV-20.02", QMON =>, QMON_ERR =>, QMON_T =>, QMON_T_CLOSE =>, QMAN_AUT =>, QREMOTE =>, QSIM =>, QLOCK =>, QERR =>, QERR_EXT =>, QwAlarm =>)
   END_RUNG
   RUNG wire#powerrail
      I_Contact( "ZSC-20.02" )
      Contact( #"AV-20.02".QCMD_OP )
   END_RUNG wire#w1
   RUNG wire#powerrail
      Contact( "ZSC-20.02" )
   END_RUNG wire#w2
   RUNG wire#powerrail
      I_Contact( #"AV-20.02".QCMD_OP )
   END_RUNG wire#w2
   // the same network as SCL:
   #"AV-20.02"(LOCK := #lock,   // "Valve"
               LIOP_SEL := #Init,
               L_AUT := #Init,
               L_REMOTE := #Init,
               L_RESET := #Reset,
               FB_OPEN := NOT "ZSC-20.02" AND #"AV-20.02".QCMD_OP,
               FB_CLOSE := "ZSC-20.02" OR NOT #"AV-20.02".QCMD_OP,
               L_MON := #Init,
               INSTANCE := 'AV-20.02',
               QCMD_OP => "AV-20.02");
END_REGION

REGION Network 3: AV-20.03
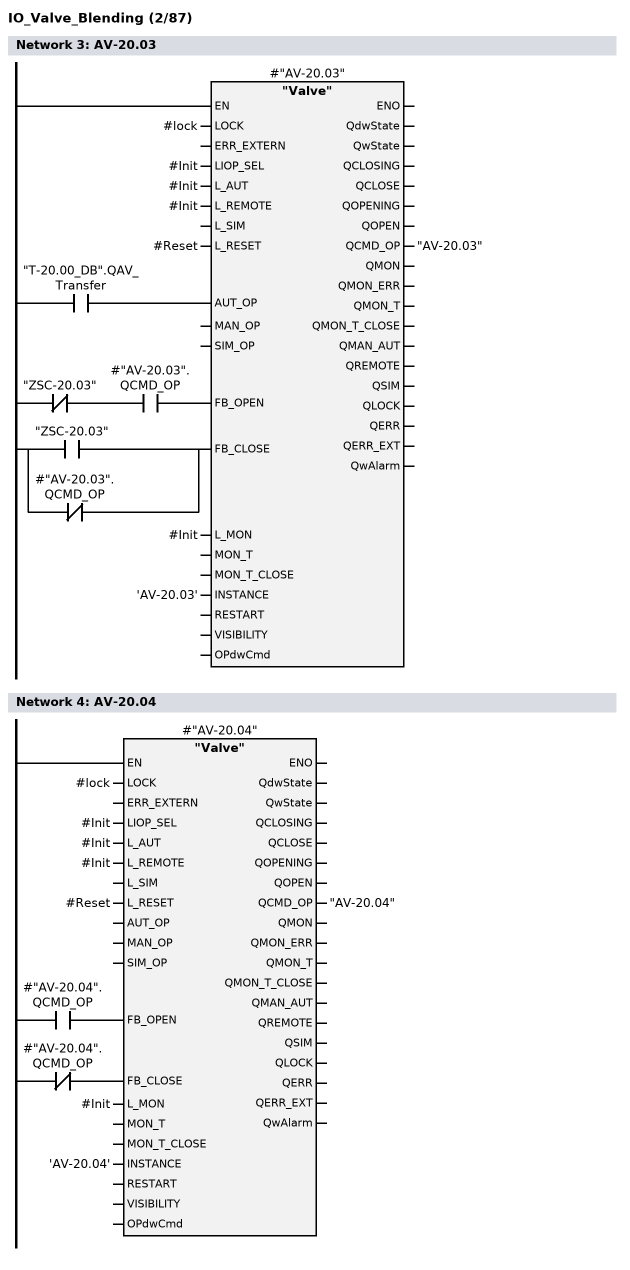
   RUNG wire#powerrail
      #"AV-20.03"(AUT_OP := wire#w1, FB_OPEN := wire#w2, FB_CLOSE := wire#w3, LOCK := #lock, ERR_EXTERN :=, LIOP_SEL := #Init, L_AUT := #Init, L_REMOTE := #Init, L_SIM :=, L_RESET := #Reset, MAN_OP :=, SIM_OP :=, L_MON := #Init, MON_T :=, MON_T_CLOSE :=, INSTANCE := 'AV-20.03', RESTART :=, VISIBILITY :=, OPdwCmd :=, QdwState =>, QwState =>, QCLOSING =>, QCLOSE =>, QOPENING =>, QOPEN =>, QCMD_OP => "AV-20.03", QMON =>, QMON_ERR =>, QMON_T =>, QMON_T_CLOSE =>, QMAN_AUT =>, QREMOTE =>, QSIM =>, QLOCK =>, QERR =>, QERR_EXT =>, QwAlarm =>)
   END_RUNG
   RUNG wire#powerrail
      Contact( "T-20.00_DB".QAV_Transfer )
   END_RUNG wire#w1
   RUNG wire#powerrail
      I_Contact( "ZSC-20.03" )
      Contact( #"AV-20.03".QCMD_OP )
   END_RUNG wire#w2
   RUNG wire#powerrail
      Contact( "ZSC-20.03" )
   END_RUNG wire#w3
   RUNG wire#powerrail
      I_Contact( #"AV-20.03".QCMD_OP )
   END_RUNG wire#w3
   // the same network as SCL:
   #"AV-20.03"(LOCK := #lock,   // "Valve"
               LIOP_SEL := #Init,
               L_AUT := #Init,
               L_REMOTE := #Init,
               L_RESET := #Reset,
               AUT_OP := "T-20.00_DB".QAV_Transfer,
               FB_OPEN := NOT "ZSC-20.03" AND #"AV-20.03".QCMD_OP,
               FB_CLOSE := "ZSC-20.03" OR NOT #"AV-20.03".QCMD_OP,
               L_MON := #Init,
               INSTANCE := 'AV-20.03',
               QCMD_OP => "AV-20.03");
END_REGION

REGION Network 4: AV-20.04
   RUNG wire#powerrail
      #"AV-20.04"(FB_OPEN := wire#w1, FB_CLOSE := wire#w2, LOCK := #lock, ERR_EXTERN :=, LIOP_SEL := #Init, L_AUT := #Init, L_REMOTE := #Init, L_SIM :=, L_RESET := #Reset, AUT_OP :=, MAN_OP :=, SIM_OP :=, L_MON := #Init, MON_T :=, MON_T_CLOSE :=, INSTANCE := 'AV-20.04', RESTART :=, VISIBILITY :=, OPdwCmd :=, QdwState =>, QwState =>, QCLOSING =>, QCLOSE =>, QOPENING =>, QOPEN =>, QCMD_OP => "AV-20.04", QMON =>, QMON_ERR =>, QMON_T =>, QMON_T_CLOSE =>, QMAN_AUT =>, QREMOTE =>, QSIM =>, QLOCK =>, QERR =>, QERR_EXT =>, QwAlarm =>)
   END_RUNG
   RUNG wire#powerrail
      Contact( #"AV-20.04".QCMD_OP )
   END_RUNG wire#w1
   RUNG wire#powerrail
      I_Contact( #"AV-20.04".QCMD_OP )
   END_RUNG wire#w2
   // the same network as SCL:
   #"AV-20.04"(LOCK := #lock,   // "Valve"
               LIOP_SEL := #Init,
               L_AUT := #Init,
               L_REMOTE := #Init,
               L_RESET := #Reset,
               FB_OPEN := #"AV-20.04".QCMD_OP,
               FB_CLOSE := NOT #"AV-20.04".QCMD_OP,
               L_MON := #Init,
               INSTANCE := 'AV-20.04',
               QCMD_OP => "AV-20.04");
END_REGION

REGION Network 5: AV-20.05
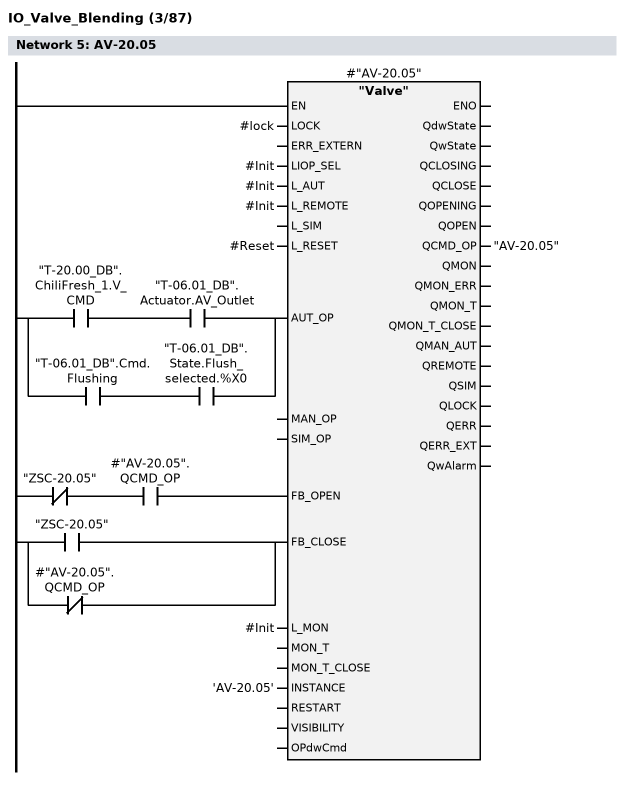
   RUNG wire#powerrail
      #"AV-20.05"(AUT_OP := wire#w1, FB_OPEN := wire#w2, FB_CLOSE := wire#w3, LOCK := #lock, ERR_EXTERN :=, LIOP_SEL := #Init, L_AUT := #Init, L_REMOTE := #Init, L_SIM :=, L_RESET := #Reset, MAN_OP :=, SIM_OP :=, L_MON := #Init, MON_T :=, MON_T_CLOSE :=, INSTANCE := 'AV-20.05', RESTART :=, VISIBILITY :=, OPdwCmd :=, QdwState =>, QwState =>, QCLOSING =>, QCLOSE =>, QOPENING =>, QOPEN =>, QCMD_OP => "AV-20.05", QMON =>, QMON_ERR =>, QMON_T =>, QMON_T_CLOSE =>, QMAN_AUT =>, QREMOTE =>, QSIM =>, QLOCK =>, QERR =>, QERR_EXT =>, QwAlarm =>)
   END_RUNG
   RUNG wire#powerrail
      Contact( "T-20.00_DB".ChiliFresh_1.V_CMD )
      Contact( "T-06.01_DB".Actuator.AV_Outlet )
   END_RUNG wire#w1
   RUNG wire#powerrail
      Contact( "T-06.01_DB".Cmd.Flushing )
      Contact( "T-06.01_DB".State.Flush_selected.%X0 )
   END_RUNG wire#w1
   RUNG wire#powerrail
      I_Contact( "ZSC-20.05" )
      Contact( #"AV-20.05".QCMD_OP )
   END_RUNG wire#w2
   RUNG wire#powerrail
      Contact( "ZSC-20.05" )
   END_RUNG wire#w3
   RUNG wire#powerrail
      I_Contact( #"AV-20.05".QCMD_OP )
   END_RUNG wire#w3
   // the same network as SCL:
   #"AV-20.05"(LOCK := #lock,   // "Valve"
               LIOP_SEL := #Init,
               L_AUT := #Init,
               L_REMOTE := #Init,
               L_RESET := #Reset,
               AUT_OP := ("T-20.00_DB".ChiliFresh_1.V_CMD AND "T-06.01_DB".Actuator.AV_Outlet) OR ("T-06.01_DB".Cmd.Flushing AND "T-06.01_DB".State.Flush_selected.%X0),
               FB_OPEN := NOT "ZSC-20.05" AND #"AV-20.05".QCMD_OP,
               FB_CLOSE := "ZSC-20.05" OR NOT #"AV-20.05".QCMD_OP,
               L_MON := #Init,
               INSTANCE := 'AV-20.05',
               QCMD_OP => "AV-20.05");
END_REGION

REGION Network 6: AV-20.06
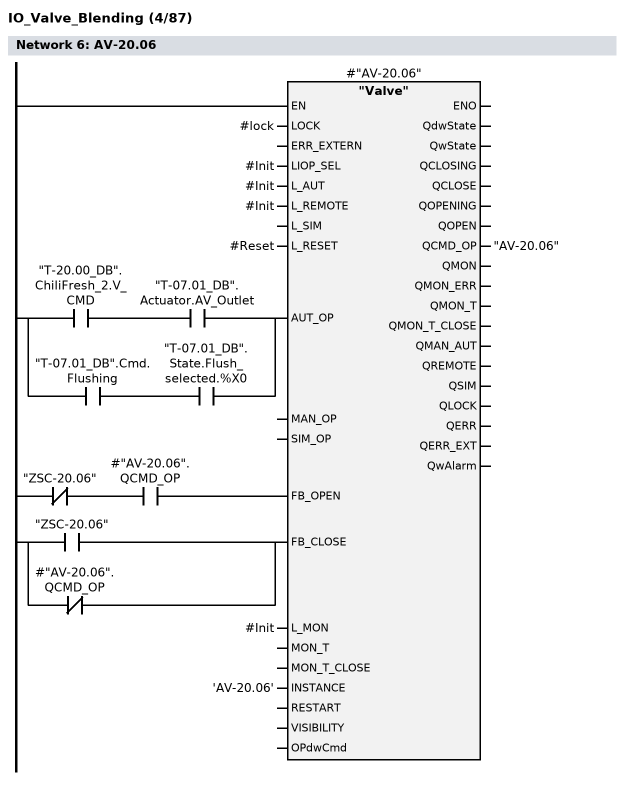
   RUNG wire#powerrail
      #"AV-20.06"(AUT_OP := wire#w1, FB_OPEN := wire#w2, FB_CLOSE := wire#w3, LOCK := #lock, ERR_EXTERN :=, LIOP_SEL := #Init, L_AUT := #Init, L_REMOTE := #Init, L_SIM :=, L_RESET := #Reset, MAN_OP :=, SIM_OP :=, L_MON := #Init, MON_T :=, MON_T_CLOSE :=, INSTANCE := 'AV-20.06', RESTART :=, VISIBILITY :=, OPdwCmd :=, QdwState =>, QwState =>, QCLOSING =>, QCLOSE =>, QOPENING =>, QOPEN =>, QCMD_OP => "AV-20.06", QMON =>, QMON_ERR =>, QMON_T =>, QMON_T_CLOSE =>, QMAN_AUT =>, QREMOTE =>, QSIM =>, QLOCK =>, QERR =>, QERR_EXT =>, QwAlarm =>)
   END_RUNG
   RUNG wire#powerrail
      Contact( "T-20.00_DB".ChiliFresh_2.V_CMD )
      Contact( "T-07.01_DB".Actuator.AV_Outlet )
   END_RUNG wire#w1
   RUNG wire#powerrail
      Contact( "T-07.01_DB".Cmd.Flushing )
      Contact( "T-07.01_DB".State.Flush_selected.%X0 )
   END_RUNG wire#w1
   RUNG wire#powerrail
      I_Contact( "ZSC-20.06" )
      Contact( #"AV-20.06".QCMD_OP )
   END_RUNG wire#w2
   RUNG wire#powerrail
      Contact( "ZSC-20.06" )
   END_RUNG wire#w3
   RUNG wire#powerrail
      I_Contact( #"AV-20.06".QCMD_OP )
   END_RUNG wire#w3
   // the same network as SCL:
   #"AV-20.06"(LOCK := #lock,   // "Valve"
               LIOP_SEL := #Init,
               L_AUT := #Init,
               L_REMOTE := #Init,
               L_RESET := #Reset,
               AUT_OP := ("T-20.00_DB".ChiliFresh_2.V_CMD AND "T-07.01_DB".Actuator.AV_Outlet) OR ("T-07.01_DB".Cmd.Flushing AND "T-07.01_DB".State.Flush_selected.%X0),
               FB_OPEN := NOT "ZSC-20.06" AND #"AV-20.06".QCMD_OP,
               FB_CLOSE := "ZSC-20.06" OR NOT #"AV-20.06".QCMD_OP,
               L_MON := #Init,
               INSTANCE := 'AV-20.06',
               QCMD_OP => "AV-20.06");
END_REGION

REGION Network 7: AV-20.07
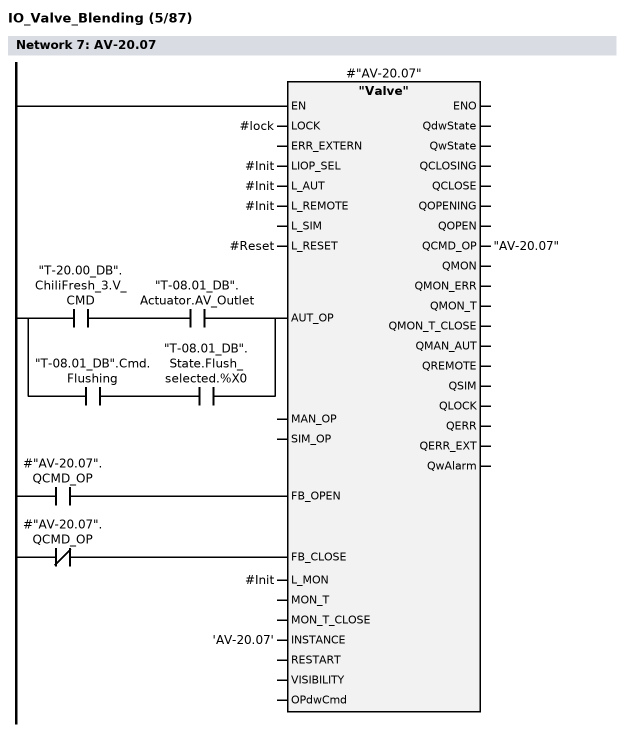
   RUNG wire#powerrail
      #"AV-20.07"(AUT_OP := wire#w1, FB_OPEN := wire#w2, FB_CLOSE := wire#w3, LOCK := #lock, ERR_EXTERN :=, LIOP_SEL := #Init, L_AUT := #Init, L_REMOTE := #Init, L_SIM :=, L_RESET := #Reset, MAN_OP :=, SIM_OP :=, L_MON := #Init, MON_T :=, MON_T_CLOSE :=, INSTANCE := 'AV-20.07', RESTART :=, VISIBILITY :=, OPdwCmd :=, QdwState =>, QwState =>, QCLOSING =>, QCLOSE =>, QOPENING =>, QOPEN =>, QCMD_OP => "AV-20.07", QMON =>, QMON_ERR =>, QMON_T =>, QMON_T_CLOSE =>, QMAN_AUT =>, QREMOTE =>, QSIM =>, QLOCK =>, QERR =>, QERR_EXT =>, QwAlarm =>)
   END_RUNG
   RUNG wire#powerrail
      Contact( "T-20.00_DB".ChiliFresh_3.V_CMD )
      Contact( "T-08.01_DB".Actuator.AV_Outlet )
   END_RUNG wire#w1
   RUNG wire#powerrail
      Contact( "T-08.01_DB".Cmd.Flushing )
      Contact( "T-08.01_DB".State.Flush_selected.%X0 )
   END_RUNG wire#w1
   RUNG wire#powerrail
      Contact( #"AV-20.07".QCMD_OP )
   END_RUNG wire#w2
   RUNG wire#powerrail
      I_Contact( #"AV-20.07".QCMD_OP )
   END_RUNG wire#w3
   // the same network as SCL:
   #"AV-20.07"(LOCK := #lock,   // "Valve"
               LIOP_SEL := #Init,
               L_AUT := #Init,
               L_REMOTE := #Init,
               L_RESET := #Reset,
               AUT_OP := ("T-20.00_DB".ChiliFresh_3.V_CMD AND "T-08.01_DB".Actuator.AV_Outlet) OR ("T-08.01_DB".Cmd.Flushing AND "T-08.01_DB".State.Flush_selected.%X0),
               FB_OPEN := #"AV-20.07".QCMD_OP,
               FB_CLOSE := NOT #"AV-20.07".QCMD_OP,
               L_MON := #Init,
               INSTANCE := 'AV-20.07',
               QCMD_OP => "AV-20.07");
END_REGION

REGION Network 8: AV-20.08
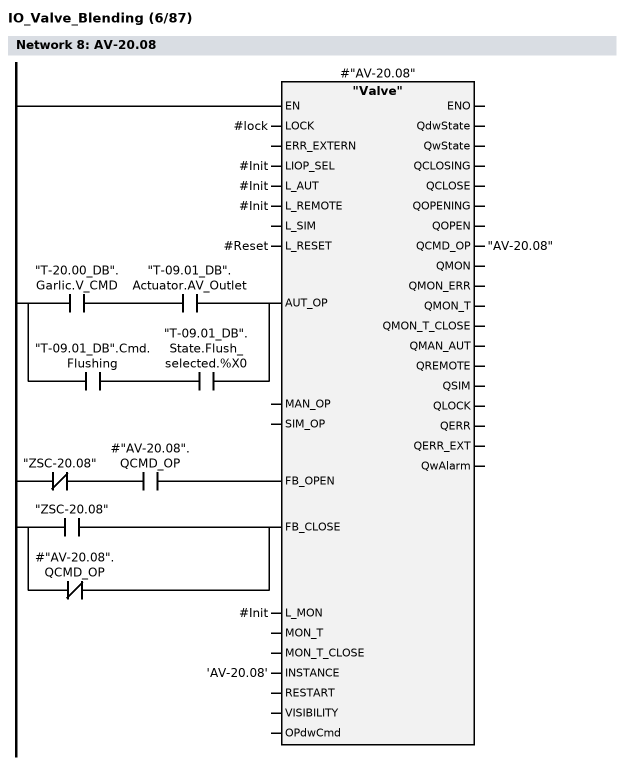
   RUNG wire#powerrail
      #"AV-20.08"(AUT_OP := wire#w1, FB_OPEN := wire#w2, FB_CLOSE := wire#w3, LOCK := #lock, ERR_EXTERN :=, LIOP_SEL := #Init, L_AUT := #Init, L_REMOTE := #Init, L_SIM :=, L_RESET := #Reset, MAN_OP :=, SIM_OP :=, L_MON := #Init, MON_T :=, MON_T_CLOSE :=, INSTANCE := 'AV-20.08', RESTART :=, VISIBILITY :=, OPdwCmd :=, QdwState =>, QwState =>, QCLOSING =>, QCLOSE =>, QOPENING =>, QOPEN =>, QCMD_OP => "AV-20.08", QMON =>, QMON_ERR =>, QMON_T =>, QMON_T_CLOSE =>, QMAN_AUT =>, QREMOTE =>, QSIM =>, QLOCK =>, QERR =>, QERR_EXT =>, QwAlarm =>)
   END_RUNG
   RUNG wire#powerrail
      Contact( "T-20.00_DB".Garlic.V_CMD )
      Contact( "T-09.01_DB".Actuator.AV_Outlet )
   END_RUNG wire#w1
   RUNG wire#powerrail
      Contact( "T-09.01_DB".Cmd.Flushing )
      Contact( "T-09.01_DB".State.Flush_selected.%X0 )
   END_RUNG wire#w1
   RUNG wire#powerrail
      I_Contact( "ZSC-20.08" )
      Contact( #"AV-20.08".QCMD_OP )
   END_RUNG wire#w2
   RUNG wire#powerrail
      Contact( "ZSC-20.08" )
   END_RUNG wire#w3
   RUNG wire#powerrail
      I_Contact( #"AV-20.08".QCMD_OP )
   END_RUNG wire#w3
   // the same network as SCL:
   #"AV-20.08"(LOCK := #lock,   // "Valve"
               LIOP_SEL := #Init,
               L_AUT := #Init,
               L_REMOTE := #Init,
               L_RESET := #Reset,
               AUT_OP := ("T-20.00_DB".Garlic.V_CMD AND "T-09.01_DB".Actuator.AV_Outlet) OR ("T-09.01_DB".Cmd.Flushing AND "T-09.01_DB".State.Flush_selected.%X0),
               FB_OPEN := NOT "ZSC-20.08" AND #"AV-20.08".QCMD_OP,
               FB_CLOSE := "ZSC-20.08" OR NOT #"AV-20.08".QCMD_OP,
               L_MON := #Init,
               INSTANCE := 'AV-20.08',
               QCMD_OP => "AV-20.08");
END_REGION

REGION Network 9: AV-20.09
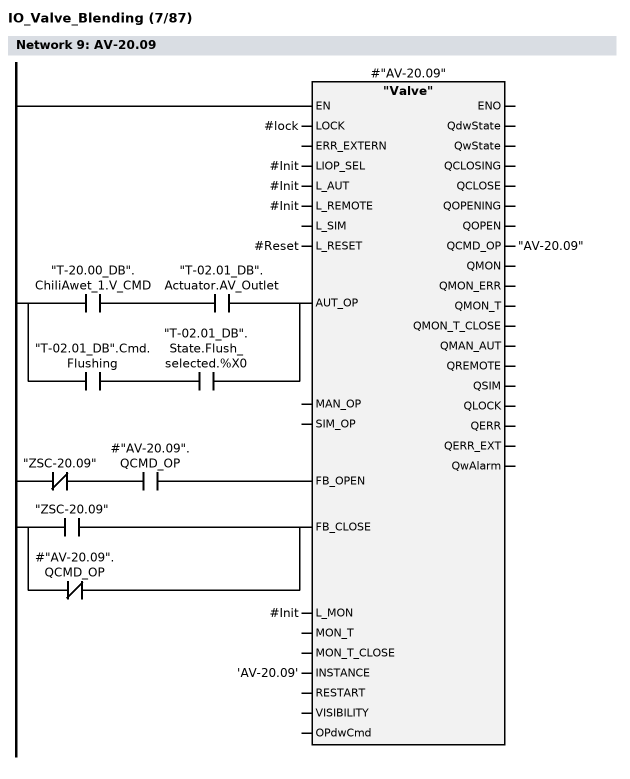
   RUNG wire#powerrail
      #"AV-20.09"(AUT_OP := wire#w1, FB_OPEN := wire#w2, FB_CLOSE := wire#w3, LOCK := #lock, ERR_EXTERN :=, LIOP_SEL := #Init, L_AUT := #Init, L_REMOTE := #Init, L_SIM :=, L_RESET := #Reset, MAN_OP :=, SIM_OP :=, L_MON := #Init, MON_T :=, MON_T_CLOSE :=, INSTANCE := 'AV-20.09', RESTART :=, VISIBILITY :=, OPdwCmd :=, QdwState =>, QwState =>, QCLOSING =>, QCLOSE =>, QOPENING =>, QOPEN =>, QCMD_OP => "AV-20.09", QMON =>, QMON_ERR =>, QMON_T =>, QMON_T_CLOSE =>, QMAN_AUT =>, QREMOTE =>, QSIM =>, QLOCK =>, QERR =>, QERR_EXT =>, QwAlarm =>)
   END_RUNG
   RUNG wire#powerrail
      Contact( "T-20.00_DB".ChiliAwet_1.V_CMD )
      Contact( "T-02.01_DB".Actuator.AV_Outlet )
   END_RUNG wire#w1
   RUNG wire#powerrail
      Contact( "T-02.01_DB".Cmd.Flushing )
      Contact( "T-02.01_DB".State.Flush_selected.%X0 )
   END_RUNG wire#w1
   RUNG wire#powerrail
      I_Contact( "ZSC-20.09" )
      Contact( #"AV-20.09".QCMD_OP )
   END_RUNG wire#w2
   RUNG wire#powerrail
      Contact( "ZSC-20.09" )
   END_RUNG wire#w3
   RUNG wire#powerrail
      I_Contact( #"AV-20.09".QCMD_OP )
   END_RUNG wire#w3
   // the same network as SCL:
   #"AV-20.09"(LOCK := #lock,   // "Valve"
               LIOP_SEL := #Init,
               L_AUT := #Init,
               L_REMOTE := #Init,
               L_RESET := #Reset,
               AUT_OP := ("T-20.00_DB".ChiliAwet_1.V_CMD AND "T-02.01_DB".Actuator.AV_Outlet) OR ("T-02.01_DB".Cmd.Flushing AND "T-02.01_DB".State.Flush_selected.%X0),
               FB_OPEN := NOT "ZSC-20.09" AND #"AV-20.09".QCMD_OP,
               FB_CLOSE := "ZSC-20.09" OR NOT #"AV-20.09".QCMD_OP,
               L_MON := #Init,
               INSTANCE := 'AV-20.09',
               QCMD_OP => "AV-20.09");
END_REGION

REGION Network 10: AV-20.10
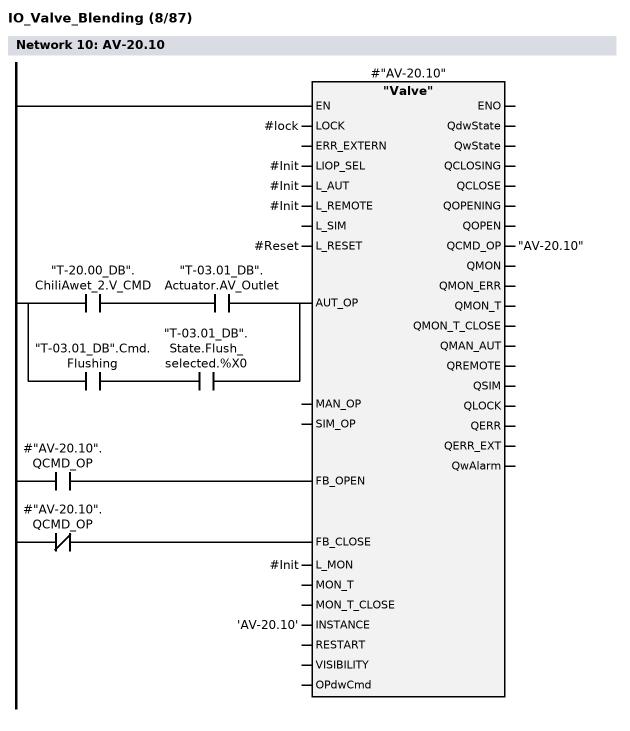
   RUNG wire#powerrail
      #"AV-20.10"(AUT_OP := wire#w1, FB_OPEN := wire#w2, FB_CLOSE := wire#w3, LOCK := #lock, ERR_EXTERN :=, LIOP_SEL := #Init, L_AUT := #Init, L_REMOTE := #Init, L_SIM :=, L_RESET := #Reset, MAN_OP :=, SIM_OP :=, L_MON := #Init, MON_T :=, MON_T_CLOSE :=, INSTANCE := 'AV-20.10', RESTART :=, VISIBILITY :=, OPdwCmd :=, QdwState =>, QwState =>, QCLOSING =>, QCLOSE =>, QOPENING =>, QOPEN =>, QCMD_OP => "AV-20.10", QMON =>, QMON_ERR =>, QMON_T =>, QMON_T_CLOSE =>, QMAN_AUT =>, QREMOTE =>, QSIM =>, QLOCK =>, QERR =>, QERR_EXT =>, QwAlarm =>)
   END_RUNG
   RUNG wire#powerrail
      Contact( "T-20.00_DB".ChiliAwet_2.V_CMD )
      Contact( "T-03.01_DB".Actuator.AV_Outlet )
   END_RUNG wire#w1
   RUNG wire#powerrail
      Contact( "T-03.01_DB".Cmd.Flushing )
      Contact( "T-03.01_DB".State.Flush_selected.%X0 )
   END_RUNG wire#w1
   RUNG wire#powerrail
      Contact( #"AV-20.10".QCMD_OP )
   END_RUNG wire#w2
   RUNG wire#powerrail
      I_Contact( #"AV-20.10".QCMD_OP )
   END_RUNG wire#w3
   // the same network as SCL:
   #"AV-20.10"(LOCK := #lock,   // "Valve"
               LIOP_SEL := #Init,
               L_AUT := #Init,
               L_REMOTE := #Init,
               L_RESET := #Reset,
               AUT_OP := ("T-20.00_DB".ChiliAwet_2.V_CMD AND "T-03.01_DB".Actuator.AV_Outlet) OR ("T-03.01_DB".Cmd.Flushing AND "T-03.01_DB".State.Flush_selected.%X0),
               FB_OPEN := #"AV-20.10".QCMD_OP,
               FB_CLOSE := NOT #"AV-20.10".QCMD_OP,
               L_MON := #Init,
               INSTANCE := 'AV-20.10',
               QCMD_OP => "AV-20.10");
END_REGION

REGION Network 11: AV-20.11
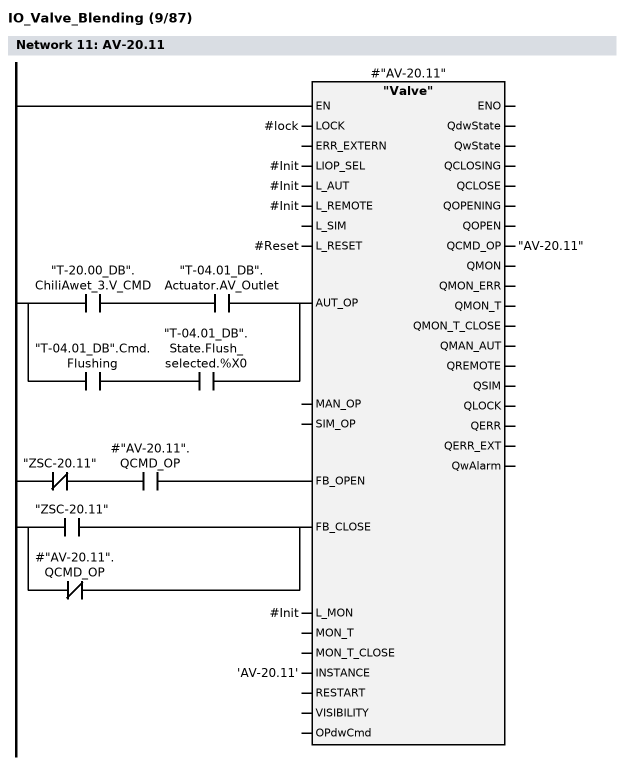
   RUNG wire#powerrail
      #"AV-20.11"(AUT_OP := wire#w1, FB_OPEN := wire#w2, FB_CLOSE := wire#w3, LOCK := #lock, ERR_EXTERN :=, LIOP_SEL := #Init, L_AUT := #Init, L_REMOTE := #Init, L_SIM :=, L_RESET := #Reset, MAN_OP :=, SIM_OP :=, L_MON := #Init, MON_T :=, MON_T_CLOSE :=, INSTANCE := 'AV-20.11', RESTART :=, VISIBILITY :=, OPdwCmd :=, QdwState =>, QwState =>, QCLOSING =>, QCLOSE =>, QOPENING =>, QOPEN =>, QCMD_OP => "AV-20.11", QMON =>, QMON_ERR =>, QMON_T =>, QMON_T_CLOSE =>, QMAN_AUT =>, QREMOTE =>, QSIM =>, QLOCK =>, QERR =>, QERR_EXT =>, QwAlarm =>)
   END_RUNG
   RUNG wire#powerrail
      Contact( "T-20.00_DB".ChiliAwet_3.V_CMD )
      Contact( "T-04.01_DB".Actuator.AV_Outlet )
   END_RUNG wire#w1
   RUNG wire#powerrail
      Contact( "T-04.01_DB".Cmd.Flushing )
      Contact( "T-04.01_DB".State.Flush_selected.%X0 )
   END_RUNG wire#w1
   RUNG wire#powerrail
      I_Contact( "ZSC-20.11" )
      Contact( #"AV-20.11".QCMD_OP )
   END_RUNG wire#w2
   RUNG wire#powerrail
      Contact( "ZSC-20.11" )
   END_RUNG wire#w3
   RUNG wire#powerrail
      I_Contact( #"AV-20.11".QCMD_OP )
   END_RUNG wire#w3
   // the same network as SCL:
   #"AV-20.11"(LOCK := #lock,   // "Valve"
               LIOP_SEL := #Init,
               L_AUT := #Init,
               L_REMOTE := #Init,
               L_RESET := #Reset,
               AUT_OP := ("T-20.00_DB".ChiliAwet_3.V_CMD AND "T-04.01_DB".Actuator.AV_Outlet) OR ("T-04.01_DB".Cmd.Flushing AND "T-04.01_DB".State.Flush_selected.%X0),
               FB_OPEN := NOT "ZSC-20.11" AND #"AV-20.11".QCMD_OP,
               FB_CLOSE := "ZSC-20.11" OR NOT #"AV-20.11".QCMD_OP,
               L_MON := #Init,
               INSTANCE := 'AV-20.11',
               QCMD_OP => "AV-20.11");
END_REGION

REGION Network 12: AV-20.12
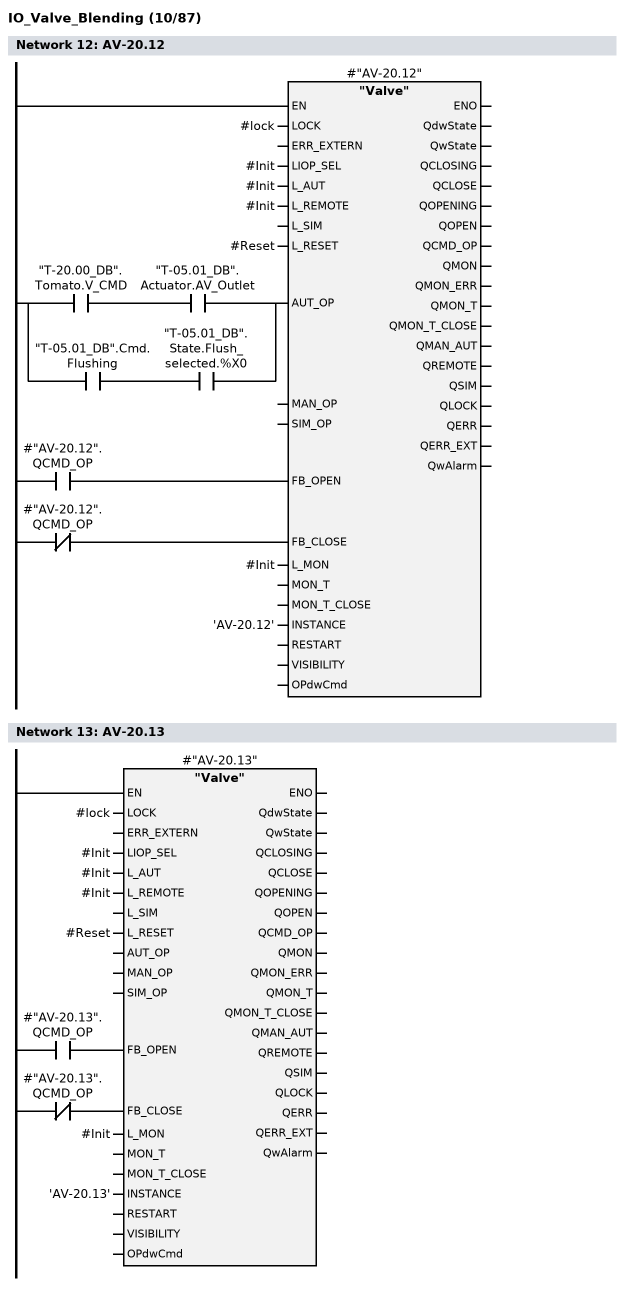
   RUNG wire#powerrail
      #"AV-20.12"(AUT_OP := wire#w1, FB_OPEN := wire#w2, FB_CLOSE := wire#w3, LOCK := #lock, ERR_EXTERN :=, LIOP_SEL := #Init, L_AUT := #Init, L_REMOTE := #Init, L_SIM :=, L_RESET := #Reset, MAN_OP :=, SIM_OP :=, L_MON := #Init, MON_T :=, MON_T_CLOSE :=, INSTANCE := 'AV-20.12', RESTART :=, VISIBILITY :=, OPdwCmd :=, QdwState =>, QwState =>, QCLOSING =>, QCLOSE =>, QOPENING =>, QOPEN =>, QCMD_OP =>, QMON =>, QMON_ERR =>, QMON_T =>, QMON_T_CLOSE =>, QMAN_AUT =>, QREMOTE =>, QSIM =>, QLOCK =>, QERR =>, QERR_EXT =>, QwAlarm =>)
   END_RUNG
   RUNG wire#powerrail
      Contact( "T-20.00_DB".Tomato.V_CMD )
      Contact( "T-05.01_DB".Actuator.AV_Outlet )
   END_RUNG wire#w1
   RUNG wire#powerrail
      Contact( "T-05.01_DB".Cmd.Flushing )
      Contact( "T-05.01_DB".State.Flush_selected.%X0 )
   END_RUNG wire#w1
   RUNG wire#powerrail
      Contact( #"AV-20.12".QCMD_OP )
   END_RUNG wire#w2
   RUNG wire#powerrail
      I_Contact( #"AV-20.12".QCMD_OP )
   END_RUNG wire#w3
   // the same network as SCL:
   #"AV-20.12"(LOCK := #lock,   // "Valve"
               LIOP_SEL := #Init,
               L_AUT := #Init,
               L_REMOTE := #Init,
               L_RESET := #Reset,
               AUT_OP := ("T-20.00_DB".Tomato.V_CMD AND "T-05.01_DB".Actuator.AV_Outlet) OR ("T-05.01_DB".Cmd.Flushing AND "T-05.01_DB".State.Flush_selected.%X0),
               FB_OPEN := #"AV-20.12".QCMD_OP,
               FB_CLOSE := NOT #"AV-20.12".QCMD_OP,
               L_MON := #Init,
               INSTANCE := 'AV-20.12');
END_REGION

REGION Network 13: AV-20.13
   RUNG wire#powerrail
      #"AV-20.13"(FB_OPEN := wire#w1, FB_CLOSE := wire#w2, LOCK := #lock, ERR_EXTERN :=, LIOP_SEL := #Init, L_AUT := #Init, L_REMOTE := #Init, L_SIM :=, L_RESET := #Reset, AUT_OP :=, MAN_OP :=, SIM_OP :=, L_MON := #Init, MON_T :=, MON_T_CLOSE :=, INSTANCE := 'AV-20.13', RESTART :=, VISIBILITY :=, OPdwCmd :=, QdwState =>, QwState =>, QCLOSING =>, QCLOSE =>, QOPENING =>, QOPEN =>, QCMD_OP =>, QMON =>, QMON_ERR =>, QMON_T =>, QMON_T_CLOSE =>, QMAN_AUT =>, QREMOTE =>, QSIM =>, QLOCK =>, QERR =>, QERR_EXT =>, QwAlarm =>)
   END_RUNG
   RUNG wire#powerrail
      Contact( #"AV-20.13".QCMD_OP )
   END_RUNG wire#w1
   RUNG wire#powerrail
      I_Contact( #"AV-20.13".QCMD_OP )
   END_RUNG wire#w2
   // the same network as SCL:
   #"AV-20.13"(LOCK := #lock,   // "Valve"
               LIOP_SEL := #Init,
               L_AUT := #Init,
               L_REMOTE := #Init,
               L_RESET := #Reset,
               FB_OPEN := #"AV-20.13".QCMD_OP,
               FB_CLOSE := NOT #"AV-20.13".QCMD_OP,
               L_MON := #Init,
               INSTANCE := 'AV-20.13');
END_REGION

REGION Network 14: AV-20.14
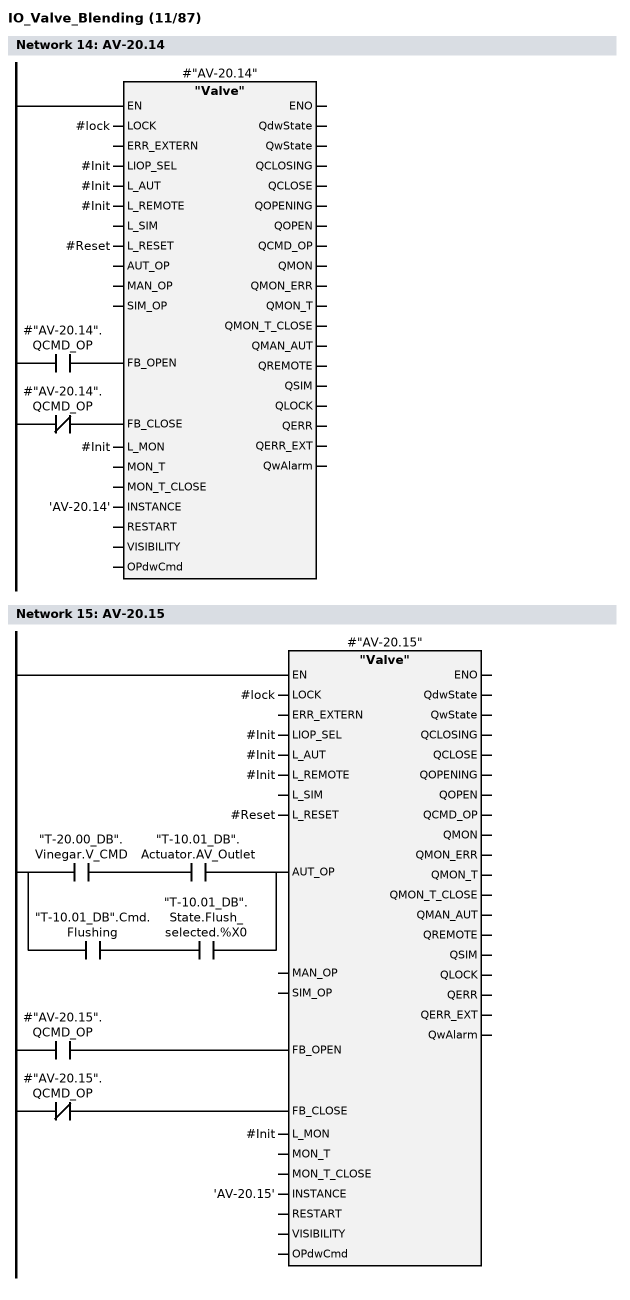
   RUNG wire#powerrail
      #"AV-20.14"(FB_OPEN := wire#w1, FB_CLOSE := wire#w2, LOCK := #lock, ERR_EXTERN :=, LIOP_SEL := #Init, L_AUT := #Init, L_REMOTE := #Init, L_SIM :=, L_RESET := #Reset, AUT_OP :=, MAN_OP :=, SIM_OP :=, L_MON := #Init, MON_T :=, MON_T_CLOSE :=, INSTANCE := 'AV-20.14', RESTART :=, VISIBILITY :=, OPdwCmd :=, QdwState =>, QwState =>, QCLOSING =>, QCLOSE =>, QOPENING =>, QOPEN =>, QCMD_OP =>, QMON =>, QMON_ERR =>, QMON_T =>, QMON_T_CLOSE =>, QMAN_AUT =>, QREMOTE =>, QSIM =>, QLOCK =>, QERR =>, QERR_EXT =>, QwAlarm =>)
   END_RUNG
   RUNG wire#powerrail
      Contact( #"AV-20.14".QCMD_OP )
   END_RUNG wire#w1
   RUNG wire#powerrail
      I_Contact( #"AV-20.14".QCMD_OP )
   END_RUNG wire#w2
   // the same network as SCL:
   #"AV-20.14"(LOCK := #lock,   // "Valve"
               LIOP_SEL := #Init,
               L_AUT := #Init,
               L_REMOTE := #Init,
               L_RESET := #Reset,
               FB_OPEN := #"AV-20.14".QCMD_OP,
               FB_CLOSE := NOT #"AV-20.14".QCMD_OP,
               L_MON := #Init,
               INSTANCE := 'AV-20.14');
END_REGION

REGION Network 15: AV-20.15
   RUNG wire#powerrail
      #"AV-20.15"(AUT_OP := wire#w1, FB_OPEN := wire#w2, FB_CLOSE := wire#w3, LOCK := #lock, ERR_EXTERN :=, LIOP_SEL := #Init, L_AUT := #Init, L_REMOTE := #Init, L_SIM :=, L_RESET := #Reset, MAN_OP :=, SIM_OP :=, L_MON := #Init, MON_T :=, MON_T_CLOSE :=, INSTANCE := 'AV-20.15', RESTART :=, VISIBILITY :=, OPdwCmd :=, QdwState =>, QwState =>, QCLOSING =>, QCLOSE =>, QOPENING =>, QOPEN =>, QCMD_OP =>, QMON =>, QMON_ERR =>, QMON_T =>, QMON_T_CLOSE =>, QMAN_AUT =>, QREMOTE =>, QSIM =>, QLOCK =>, QERR =>, QERR_EXT =>, QwAlarm =>)
   END_RUNG
   RUNG wire#powerrail
      Contact( "T-20.00_DB".Vinegar.V_CMD )
      Contact( "T-10.01_DB".Actuator.AV_Outlet )
   END_RUNG wire#w1
   RUNG wire#powerrail
      Contact( "T-10.01_DB".Cmd.Flushing )
      Contact( "T-10.01_DB".State.Flush_selected.%X0 )
   END_RUNG wire#w1
   RUNG wire#powerrail
      Contact( #"AV-20.15".QCMD_OP )
   END_RUNG wire#w2
   RUNG wire#powerrail
      I_Contact( #"AV-20.15".QCMD_OP )
   END_RUNG wire#w3
   // the same network as SCL:
   #"AV-20.15"(LOCK := #lock,   // "Valve"
               LIOP_SEL := #Init,
               L_AUT := #Init,
               L_REMOTE := #Init,
               L_RESET := #Reset,
               AUT_OP := ("T-20.00_DB".Vinegar.V_CMD AND "T-10.01_DB".Actuator.AV_Outlet) OR ("T-10.01_DB".Cmd.Flushing AND "T-10.01_DB".State.Flush_selected.%X0),
               FB_OPEN := #"AV-20.15".QCMD_OP,
               FB_CLOSE := NOT #"AV-20.15".QCMD_OP,
               L_MON := #Init,
               INSTANCE := 'AV-20.15');
END_REGION

REGION Network 16: AV-20.16
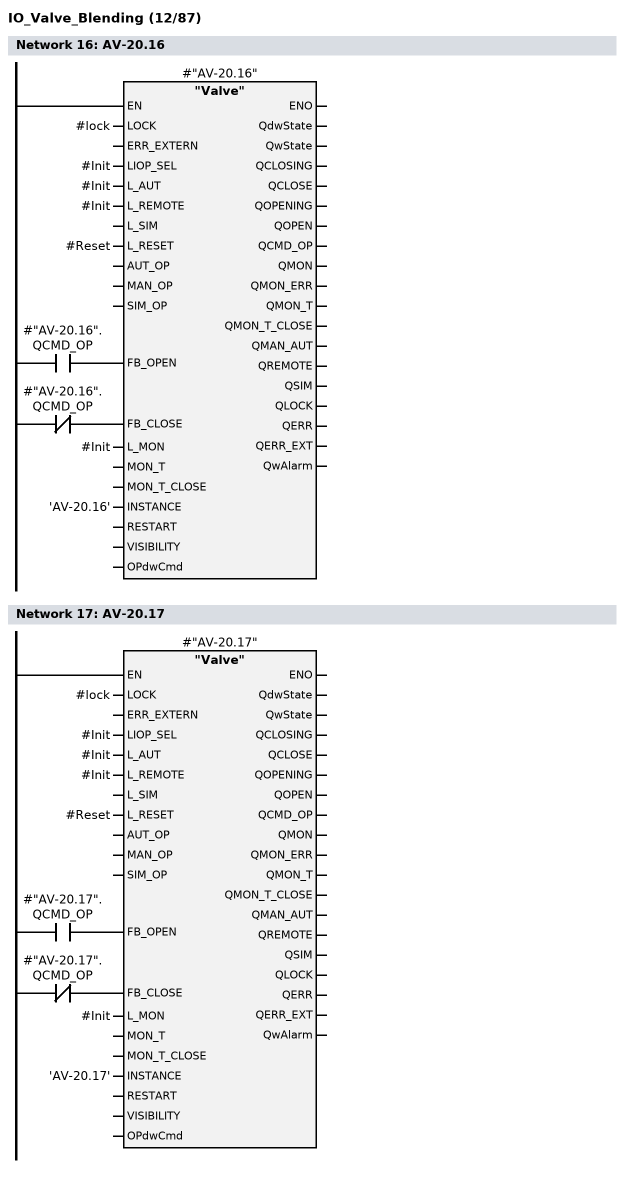
   RUNG wire#powerrail
      #"AV-20.16"(FB_OPEN := wire#w1, FB_CLOSE := wire#w2, LOCK := #lock, ERR_EXTERN :=, LIOP_SEL := #Init, L_AUT := #Init, L_REMOTE := #Init, L_SIM :=, L_RESET := #Reset, AUT_OP :=, MAN_OP :=, SIM_OP :=, L_MON := #Init, MON_T :=, MON_T_CLOSE :=, INSTANCE := 'AV-20.16', RESTART :=, VISIBILITY :=, OPdwCmd :=, QdwState =>, QwState =>, QCLOSING =>, QCLOSE =>, QOPENING =>, QOPEN =>, QCMD_OP =>, QMON =>, QMON_ERR =>, QMON_T =>, QMON_T_CLOSE =>, QMAN_AUT =>, QREMOTE =>, QSIM =>, QLOCK =>, QERR =>, QERR_EXT =>, QwAlarm =>)
   END_RUNG
   RUNG wire#powerrail
      Contact( #"AV-20.16".QCMD_OP )
   END_RUNG wire#w1
   RUNG wire#powerrail
      I_Contact( #"AV-20.16".QCMD_OP )
   END_RUNG wire#w2
   // the same network as SCL:
   #"AV-20.16"(LOCK := #lock,   // "Valve"
               LIOP_SEL := #Init,
               L_AUT := #Init,
               L_REMOTE := #Init,
               L_RESET := #Reset,
               FB_OPEN := #"AV-20.16".QCMD_OP,
               FB_CLOSE := NOT #"AV-20.16".QCMD_OP,
               L_MON := #Init,
               INSTANCE := 'AV-20.16');
END_REGION

REGION Network 17: AV-20.17
   RUNG wire#powerrail
      #"AV-20.17"(FB_OPEN := wire#w1, FB_CLOSE := wire#w2, LOCK := #lock, ERR_EXTERN :=, LIOP_SEL := #Init, L_AUT := #Init, L_REMOTE := #Init, L_SIM :=, L_RESET := #Reset, AUT_OP :=, MAN_OP :=, SIM_OP :=, L_MON := #Init, MON_T :=, MON_T_CLOSE :=, INSTANCE := 'AV-20.17', RESTART :=, VISIBILITY :=, OPdwCmd :=, QdwState =>, QwState =>, QCLOSING =>, QCLOSE =>, QOPENING =>, QOPEN =>, QCMD_OP =>, QMON =>, QMON_ERR =>, QMON_T =>, QMON_T_CLOSE =>, QMAN_AUT =>, QREMOTE =>, QSIM =>, QLOCK =>, QERR =>, QERR_EXT =>, QwAlarm =>)
   END_RUNG
   RUNG wire#powerrail
      Contact( #"AV-20.17".QCMD_OP )
   END_RUNG wire#w1
   RUNG wire#powerrail
      I_Contact( #"AV-20.17".QCMD_OP )
   END_RUNG wire#w2
   // the same network as SCL:
   #"AV-20.17"(LOCK := #lock,   // "Valve"
               LIOP_SEL := #Init,
               L_AUT := #Init,
               L_REMOTE := #Init,
               L_RESET := #Reset,
               FB_OPEN := #"AV-20.17".QCMD_OP,
               FB_CLOSE := NOT #"AV-20.17".QCMD_OP,
               L_MON := #Init,
               INSTANCE := 'AV-20.17');
END_REGION

REGION Network 18: AV-20.31
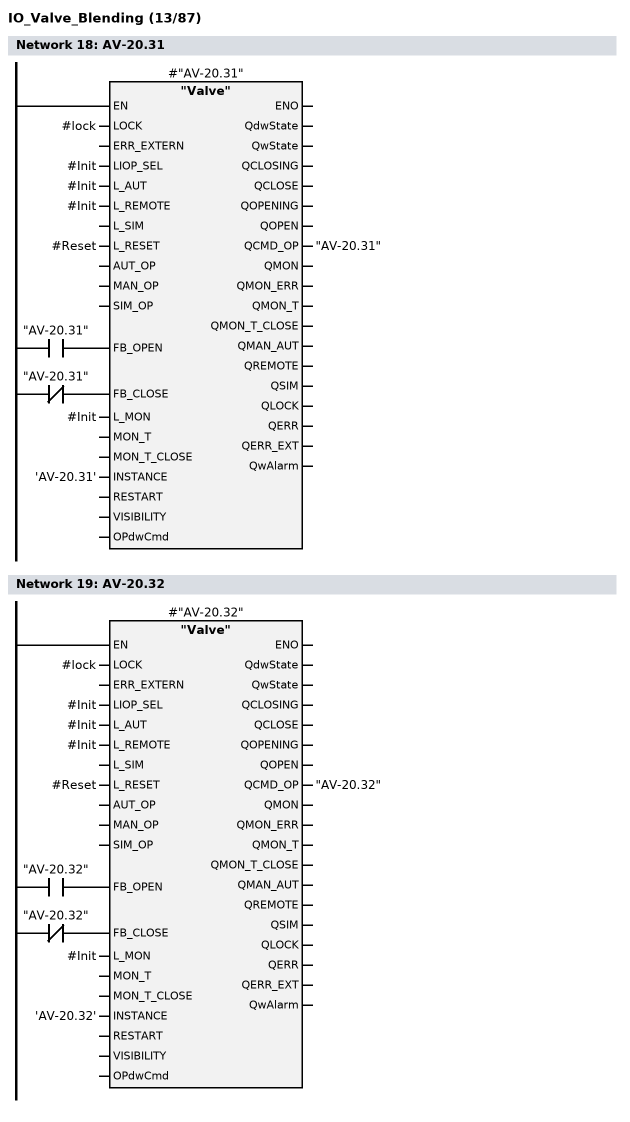
   RUNG wire#powerrail
      #"AV-20.31"(FB_OPEN := wire#w1, FB_CLOSE := wire#w2, LOCK := #lock, ERR_EXTERN :=, LIOP_SEL := #Init, L_AUT := #Init, L_REMOTE := #Init, L_SIM :=, L_RESET := #Reset, AUT_OP :=, MAN_OP :=, SIM_OP :=, L_MON := #Init, MON_T :=, MON_T_CLOSE :=, INSTANCE := 'AV-20.31', RESTART :=, VISIBILITY :=, OPdwCmd :=, QdwState =>, QwState =>, QCLOSING =>, QCLOSE =>, QOPENING =>, QOPEN =>, QCMD_OP => "AV-20.31", QMON =>, QMON_ERR =>, QMON_T =>, QMON_T_CLOSE =>, QMAN_AUT =>, QREMOTE =>, QSIM =>, QLOCK =>, QERR =>, QERR_EXT =>, QwAlarm =>)
   END_RUNG
   RUNG wire#powerrail
      Contact( "AV-20.31" )
   END_RUNG wire#w1
   RUNG wire#powerrail
      I_Contact( "AV-20.31" )
   END_RUNG wire#w2
   // the same network as SCL:
   #"AV-20.31"(LOCK := #lock,   // "Valve"
               LIOP_SEL := #Init,
               L_AUT := #Init,
               L_REMOTE := #Init,
               L_RESET := #Reset,
               FB_OPEN := "AV-20.31",
               FB_CLOSE := NOT "AV-20.31",
               L_MON := #Init,
               INSTANCE := 'AV-20.31',
               QCMD_OP => "AV-20.31");
END_REGION

REGION Network 19: AV-20.32
   RUNG wire#powerrail
      #"AV-20.32"(FB_OPEN := wire#w1, FB_CLOSE := wire#w2, LOCK := #lock, ERR_EXTERN :=, LIOP_SEL := #Init, L_AUT := #Init, L_REMOTE := #Init, L_SIM :=, L_RESET := #Reset, AUT_OP :=, MAN_OP :=, SIM_OP :=, L_MON := #Init, MON_T :=, MON_T_CLOSE :=, INSTANCE := 'AV-20.32', RESTART :=, VISIBILITY :=, OPdwCmd :=, QdwState =>, QwState =>, QCLOSING =>, QCLOSE =>, QOPENING =>, QOPEN =>, QCMD_OP => "AV-20.32", QMON =>, QMON_ERR =>, QMON_T =>, QMON_T_CLOSE =>, QMAN_AUT =>, QREMOTE =>, QSIM =>, QLOCK =>, QERR =>, QERR_EXT =>, QwAlarm =>)
   END_RUNG
   RUNG wire#powerrail
      Contact( "AV-20.32" )
   END_RUNG wire#w1
   RUNG wire#powerrail
      I_Contact( "AV-20.32" )
   END_RUNG wire#w2
   // the same network as SCL:
   #"AV-20.32"(LOCK := #lock,   // "Valve"
               LIOP_SEL := #Init,
               L_AUT := #Init,
               L_REMOTE := #Init,
               L_RESET := #Reset,
               FB_OPEN := "AV-20.32",
               FB_CLOSE := NOT "AV-20.32",
               L_MON := #Init,
               INSTANCE := 'AV-20.32',
               QCMD_OP => "AV-20.32");
END_REGION

REGION Network 20: AV-20.33
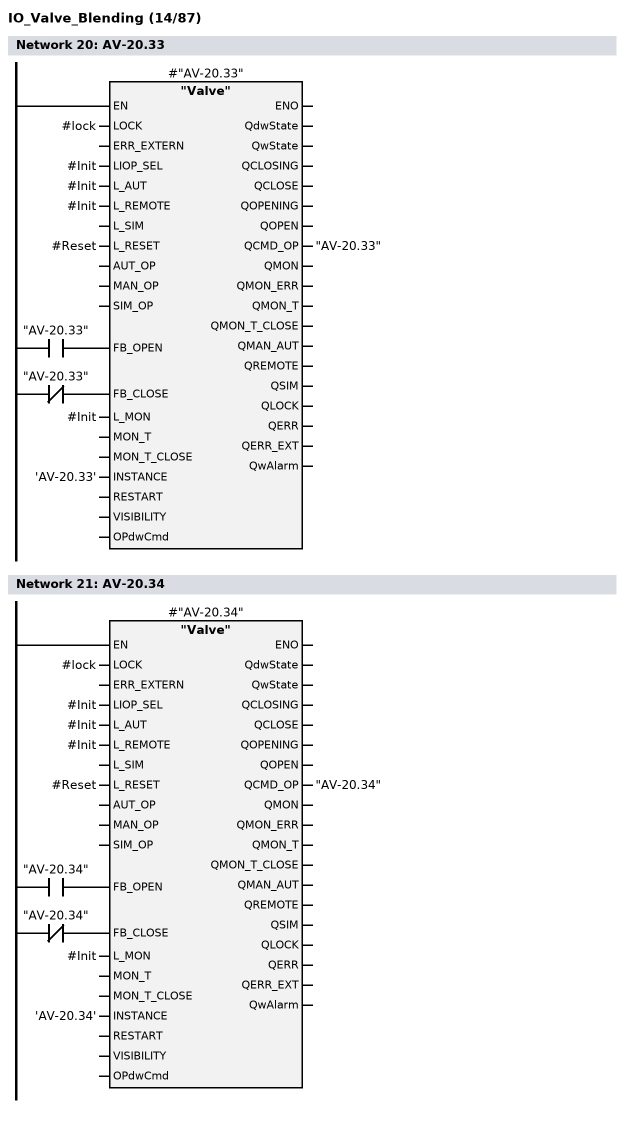
   RUNG wire#powerrail
      #"AV-20.33"(FB_OPEN := wire#w1, FB_CLOSE := wire#w2, LOCK := #lock, ERR_EXTERN :=, LIOP_SEL := #Init, L_AUT := #Init, L_REMOTE := #Init, L_SIM :=, L_RESET := #Reset, AUT_OP :=, MAN_OP :=, SIM_OP :=, L_MON := #Init, MON_T :=, MON_T_CLOSE :=, INSTANCE := 'AV-20.33', RESTART :=, VISIBILITY :=, OPdwCmd :=, QdwState =>, QwState =>, QCLOSING =>, QCLOSE =>, QOPENING =>, QOPEN =>, QCMD_OP => "AV-20.33", QMON =>, QMON_ERR =>, QMON_T =>, QMON_T_CLOSE =>, QMAN_AUT =>, QREMOTE =>, QSIM =>, QLOCK =>, QERR =>, QERR_EXT =>, QwAlarm =>)
   END_RUNG
   RUNG wire#powerrail
      Contact( "AV-20.33" )
   END_RUNG wire#w1
   RUNG wire#powerrail
      I_Contact( "AV-20.33" )
   END_RUNG wire#w2
   // the same network as SCL:
   #"AV-20.33"(LOCK := #lock,   // "Valve"
               LIOP_SEL := #Init,
               L_AUT := #Init,
               L_REMOTE := #Init,
               L_RESET := #Reset,
               FB_OPEN := "AV-20.33",
               FB_CLOSE := NOT "AV-20.33",
               L_MON := #Init,
               INSTANCE := 'AV-20.33',
               QCMD_OP => "AV-20.33");
END_REGION

REGION Network 21: AV-20.34
   RUNG wire#powerrail
      #"AV-20.34"(FB_OPEN := wire#w1, FB_CLOSE := wire#w2, LOCK := #lock, ERR_EXTERN :=, LIOP_SEL := #Init, L_AUT := #Init, L_REMOTE := #Init, L_SIM :=, L_RESET := #Reset, AUT_OP :=, MAN_OP :=, SIM_OP :=, L_MON := #Init, MON_T :=, MON_T_CLOSE :=, INSTANCE := 'AV-20.34', RESTART :=, VISIBILITY :=, OPdwCmd :=, QdwState =>, QwState =>, QCLOSING =>, QCLOSE =>, QOPENING =>, QOPEN =>, QCMD_OP => "AV-20.34", QMON =>, QMON_ERR =>, QMON_T =>, QMON_T_CLOSE =>, QMAN_AUT =>, QREMOTE =>, QSIM =>, QLOCK =>, QERR =>, QERR_EXT =>, QwAlarm =>)
   END_RUNG
   RUNG wire#powerrail
      Contact( "AV-20.34" )
   END_RUNG wire#w1
   RUNG wire#powerrail
      I_Contact( "AV-20.34" )
   END_RUNG wire#w2
   // the same network as SCL:
   #"AV-20.34"(LOCK := #lock,   // "Valve"
               LIOP_SEL := #Init,
               L_AUT := #Init,
               L_REMOTE := #Init,
               L_RESET := #Reset,
               FB_OPEN := "AV-20.34",
               FB_CLOSE := NOT "AV-20.34",
               L_MON := #Init,
               INSTANCE := 'AV-20.34',
               QCMD_OP => "AV-20.34");
END_REGION

REGION Network 22: AV-20.35
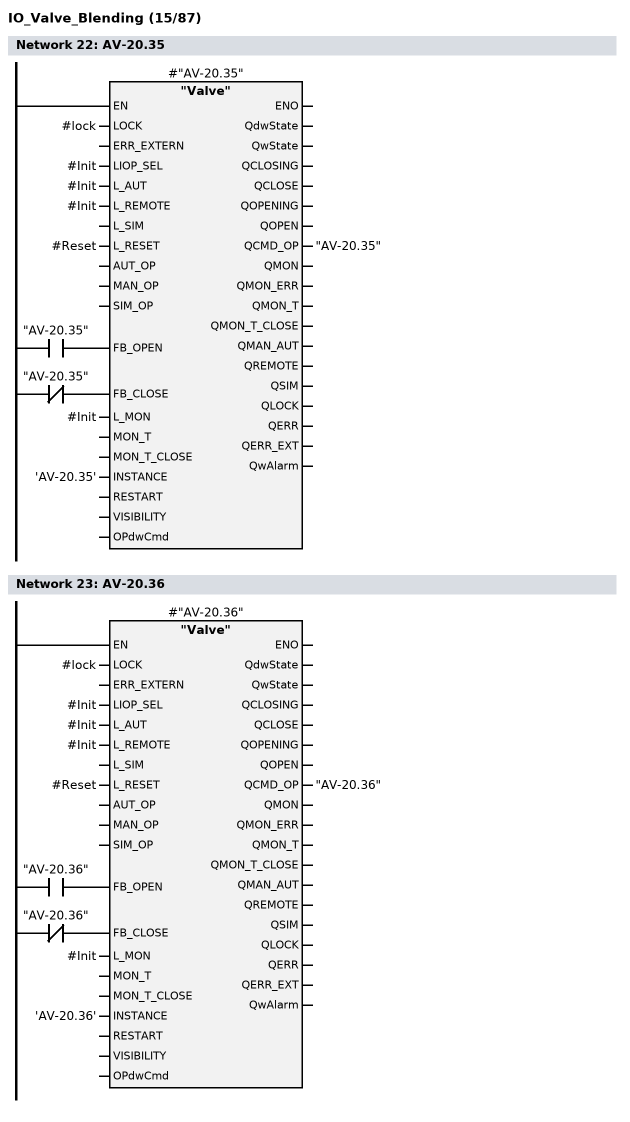
   RUNG wire#powerrail
      #"AV-20.35"(FB_OPEN := wire#w1, FB_CLOSE := wire#w2, LOCK := #lock, ERR_EXTERN :=, LIOP_SEL := #Init, L_AUT := #Init, L_REMOTE := #Init, L_SIM :=, L_RESET := #Reset, AUT_OP :=, MAN_OP :=, SIM_OP :=, L_MON := #Init, MON_T :=, MON_T_CLOSE :=, INSTANCE := 'AV-20.35', RESTART :=, VISIBILITY :=, OPdwCmd :=, QdwState =>, QwState =>, QCLOSING =>, QCLOSE =>, QOPENING =>, QOPEN =>, QCMD_OP => "AV-20.35", QMON =>, QMON_ERR =>, QMON_T =>, QMON_T_CLOSE =>, QMAN_AUT =>, QREMOTE =>, QSIM =>, QLOCK =>, QERR =>, QERR_EXT =>, QwAlarm =>)
   END_RUNG
   RUNG wire#powerrail
      Contact( "AV-20.35" )
   END_RUNG wire#w1
   RUNG wire#powerrail
      I_Contact( "AV-20.35" )
   END_RUNG wire#w2
   // the same network as SCL:
   #"AV-20.35"(LOCK := #lock,   // "Valve"
               LIOP_SEL := #Init,
               L_AUT := #Init,
               L_REMOTE := #Init,
               L_RESET := #Reset,
               FB_OPEN := "AV-20.35",
               FB_CLOSE := NOT "AV-20.35",
               L_MON := #Init,
               INSTANCE := 'AV-20.35',
               QCMD_OP => "AV-20.35");
END_REGION

REGION Network 23: AV-20.36
   RUNG wire#powerrail
      #"AV-20.36"(FB_OPEN := wire#w1, FB_CLOSE := wire#w2, LOCK := #lock, ERR_EXTERN :=, LIOP_SEL := #Init, L_AUT := #Init, L_REMOTE := #Init, L_SIM :=, L_RESET := #Reset, AUT_OP :=, MAN_OP :=, SIM_OP :=, L_MON := #Init, MON_T :=, MON_T_CLOSE :=, INSTANCE := 'AV-20.36', RESTART :=, VISIBILITY :=, OPdwCmd :=, QdwState =>, QwState =>, QCLOSING =>, QCLOSE =>, QOPENING =>, QOPEN =>, QCMD_OP => "AV-20.36", QMON =>, QMON_ERR =>, QMON_T =>, QMON_T_CLOSE =>, QMAN_AUT =>, QREMOTE =>, QSIM =>, QLOCK =>, QERR =>, QERR_EXT =>, QwAlarm =>)
   END_RUNG
   RUNG wire#powerrail
      Contact( "AV-20.36" )
   END_RUNG wire#w1
   RUNG wire#powerrail
      I_Contact( "AV-20.36" )
   END_RUNG wire#w2
   // the same network as SCL:
   #"AV-20.36"(LOCK := #lock,   // "Valve"
               LIOP_SEL := #Init,
               L_AUT := #Init,
               L_REMOTE := #Init,
               L_RESET := #Reset,
               FB_OPEN := "AV-20.36",
               FB_CLOSE := NOT "AV-20.36",
               L_MON := #Init,
               INSTANCE := 'AV-20.36',
               QCMD_OP => "AV-20.36");
END_REGION

REGION Network 24: AV-20.37
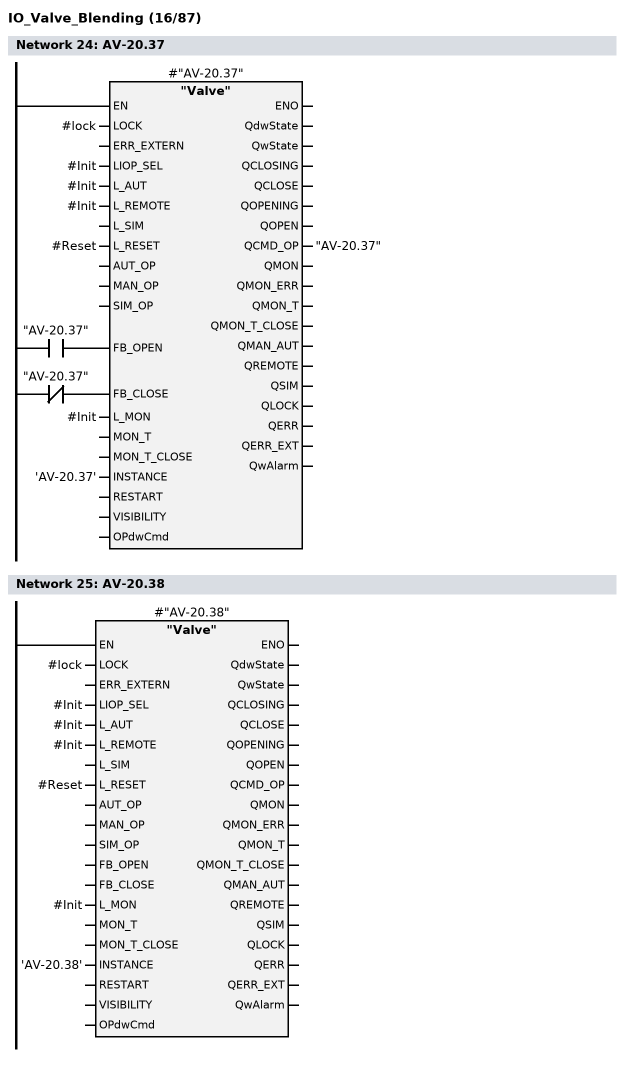
   RUNG wire#powerrail
      #"AV-20.37"(FB_OPEN := wire#w1, FB_CLOSE := wire#w2, LOCK := #lock, ERR_EXTERN :=, LIOP_SEL := #Init, L_AUT := #Init, L_REMOTE := #Init, L_SIM :=, L_RESET := #Reset, AUT_OP :=, MAN_OP :=, SIM_OP :=, L_MON := #Init, MON_T :=, MON_T_CLOSE :=, INSTANCE := 'AV-20.37', RESTART :=, VISIBILITY :=, OPdwCmd :=, QdwState =>, QwState =>, QCLOSING =>, QCLOSE =>, QOPENING =>, QOPEN =>, QCMD_OP => "AV-20.37", QMON =>, QMON_ERR =>, QMON_T =>, QMON_T_CLOSE =>, QMAN_AUT =>, QREMOTE =>, QSIM =>, QLOCK =>, QERR =>, QERR_EXT =>, QwAlarm =>)
   END_RUNG
   RUNG wire#powerrail
      Contact( "AV-20.37" )
   END_RUNG wire#w1
   RUNG wire#powerrail
      I_Contact( "AV-20.37" )
   END_RUNG wire#w2
   // the same network as SCL:
   #"AV-20.37"(LOCK := #lock,   // "Valve"
               LIOP_SEL := #Init,
               L_AUT := #Init,
               L_REMOTE := #Init,
               L_RESET := #Reset,
               FB_OPEN := "AV-20.37",
               FB_CLOSE := NOT "AV-20.37",
               L_MON := #Init,
               INSTANCE := 'AV-20.37',
               QCMD_OP => "AV-20.37");
END_REGION

REGION Network 25: AV-20.38
   RUNG wire#powerrail
      #"AV-20.38"(LOCK := #lock, ERR_EXTERN :=, LIOP_SEL := #Init, L_AUT := #Init, L_REMOTE := #Init, L_SIM :=, L_RESET := #Reset, AUT_OP :=, MAN_OP :=, SIM_OP :=, FB_OPEN :=, FB_CLOSE :=, L_MON := #Init, MON_T :=, MON_T_CLOSE :=, INSTANCE := 'AV-20.38', RESTART :=, VISIBILITY :=, OPdwCmd :=, QdwState =>, QwState =>, QCLOSING =>, QCLOSE =>, QOPENING =>, QOPEN =>, QCMD_OP =>, QMON =>, QMON_ERR =>, QMON_T =>, QMON_T_CLOSE =>, QMAN_AUT =>, QREMOTE =>, QSIM =>, QLOCK =>, QERR =>, QERR_EXT =>, QwAlarm =>)
   END_RUNG
   // the same network as SCL:
   #"AV-20.38"(LOCK := #lock,   // "Valve"
               LIOP_SEL := #Init,
               L_AUT := #Init,
               L_REMOTE := #Init,
               L_RESET := #Reset,
               L_MON := #Init,
               INSTANCE := 'AV-20.38');
END_REGION

REGION Network 26: AV-20.39
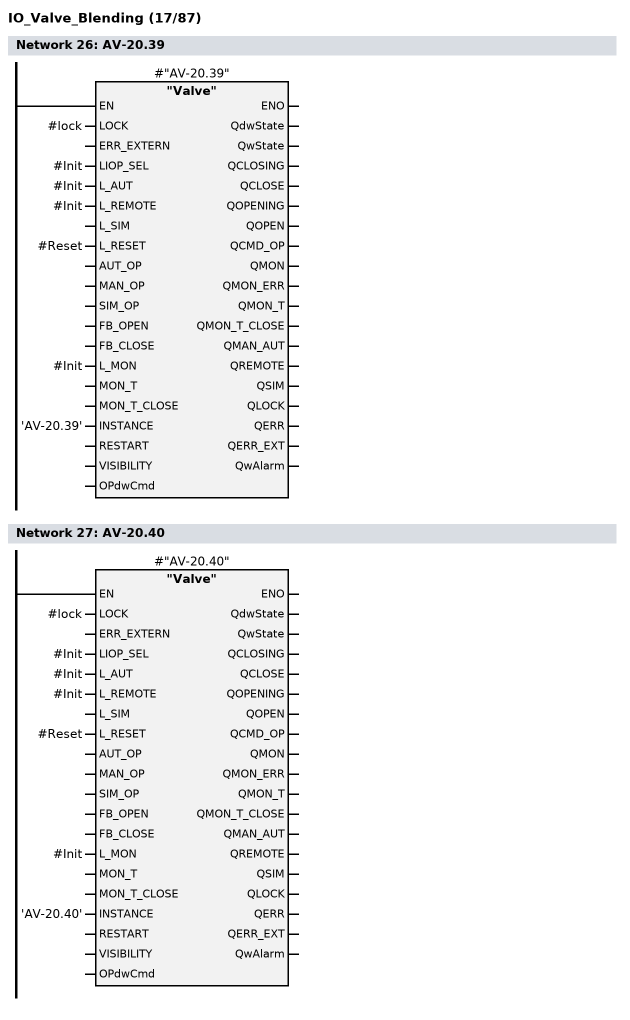
   RUNG wire#powerrail
      #"AV-20.39"(LOCK := #lock, ERR_EXTERN :=, LIOP_SEL := #Init, L_AUT := #Init, L_REMOTE := #Init, L_SIM :=, L_RESET := #Reset, AUT_OP :=, MAN_OP :=, SIM_OP :=, FB_OPEN :=, FB_CLOSE :=, L_MON := #Init, MON_T :=, MON_T_CLOSE :=, INSTANCE := 'AV-20.39', RESTART :=, VISIBILITY :=, OPdwCmd :=, QdwState =>, QwState =>, QCLOSING =>, QCLOSE =>, QOPENING =>, QOPEN =>, QCMD_OP =>, QMON =>, QMON_ERR =>, QMON_T =>, QMON_T_CLOSE =>, QMAN_AUT =>, QREMOTE =>, QSIM =>, QLOCK =>, QERR =>, QERR_EXT =>, QwAlarm =>)
   END_RUNG
   // the same network as SCL:
   #"AV-20.39"(LOCK := #lock,   // "Valve"
               LIOP_SEL := #Init,
               L_AUT := #Init,
               L_REMOTE := #Init,
               L_RESET := #Reset,
               L_MON := #Init,
               INSTANCE := 'AV-20.39');
END_REGION

REGION Network 27: AV-20.40
   RUNG wire#powerrail
      #"AV-20.40"(LOCK := #lock, ERR_EXTERN :=, LIOP_SEL := #Init, L_AUT := #Init, L_REMOTE := #Init, L_SIM :=, L_RESET := #Reset, AUT_OP :=, MAN_OP :=, SIM_OP :=, FB_OPEN :=, FB_CLOSE :=, L_MON := #Init, MON_T :=, MON_T_CLOSE :=, INSTANCE := 'AV-20.40', RESTART :=, VISIBILITY :=, OPdwCmd :=, QdwState =>, QwState =>, QCLOSING =>, QCLOSE =>, QOPENING =>, QOPEN =>, QCMD_OP =>, QMON =>, QMON_ERR =>, QMON_T =>, QMON_T_CLOSE =>, QMAN_AUT =>, QREMOTE =>, QSIM =>, QLOCK =>, QERR =>, QERR_EXT =>, QwAlarm =>)
   END_RUNG
   // the same network as SCL:
   #"AV-20.40"(LOCK := #lock,   // "Valve"
               LIOP_SEL := #Init,
               L_AUT := #Init,
               L_REMOTE := #Init,
               L_RESET := #Reset,
               L_MON := #Init,
               INSTANCE := 'AV-20.40');
END_REGION

REGION Network 28: AV-20.41
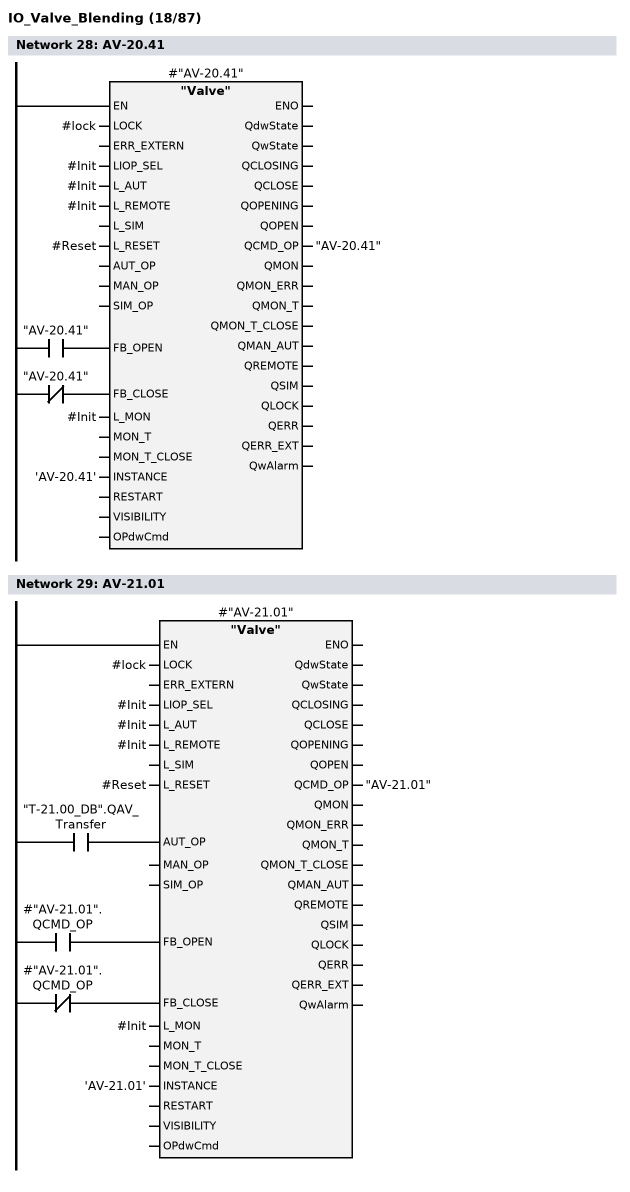
   RUNG wire#powerrail
      #"AV-20.41"(FB_OPEN := wire#w1, FB_CLOSE := wire#w2, LOCK := #lock, ERR_EXTERN :=, LIOP_SEL := #Init, L_AUT := #Init, L_REMOTE := #Init, L_SIM :=, L_RESET := #Reset, AUT_OP :=, MAN_OP :=, SIM_OP :=, L_MON := #Init, MON_T :=, MON_T_CLOSE :=, INSTANCE := 'AV-20.41', RESTART :=, VISIBILITY :=, OPdwCmd :=, QdwState =>, QwState =>, QCLOSING =>, QCLOSE =>, QOPENING =>, QOPEN =>, QCMD_OP => "AV-20.41", QMON =>, QMON_ERR =>, QMON_T =>, QMON_T_CLOSE =>, QMAN_AUT =>, QREMOTE =>, QSIM =>, QLOCK =>, QERR =>, QERR_EXT =>, QwAlarm =>)
   END_RUNG
   RUNG wire#powerrail
      Contact( "AV-20.41" )
   END_RUNG wire#w1
   RUNG wire#powerrail
      I_Contact( "AV-20.41" )
   END_RUNG wire#w2
   // the same network as SCL:
   #"AV-20.41"(LOCK := #lock,   // "Valve"
               LIOP_SEL := #Init,
               L_AUT := #Init,
               L_REMOTE := #Init,
               L_RESET := #Reset,
               FB_OPEN := "AV-20.41",
               FB_CLOSE := NOT "AV-20.41",
               L_MON := #Init,
               INSTANCE := 'AV-20.41',
               QCMD_OP => "AV-20.41");
END_REGION

REGION Network 29: AV-21.01
   RUNG wire#powerrail
      #"AV-21.01"(AUT_OP := wire#w1, FB_OPEN := wire#w2, FB_CLOSE := wire#w3, LOCK := #lock, ERR_EXTERN :=, LIOP_SEL := #Init, L_AUT := #Init, L_REMOTE := #Init, L_SIM :=, L_RESET := #Reset, MAN_OP :=, SIM_OP :=, L_MON := #Init, MON_T :=, MON_T_CLOSE :=, INSTANCE := 'AV-21.01', RESTART :=, VISIBILITY :=, OPdwCmd :=, QdwState =>, QwState =>, QCLOSING =>, QCLOSE =>, QOPENING =>, QOPEN =>, QCMD_OP => "AV-21.01", QMON =>, QMON_ERR =>, QMON_T =>, QMON_T_CLOSE =>, QMAN_AUT =>, QREMOTE =>, QSIM =>, QLOCK =>, QERR =>, QERR_EXT =>, QwAlarm =>)
   END_RUNG
   RUNG wire#powerrail
      Contact( "T-21.00_DB".QAV_Transfer )
   END_RUNG wire#w1
   RUNG wire#powerrail
      Contact( #"AV-21.01".QCMD_OP )
   END_RUNG wire#w2
   RUNG wire#powerrail
      I_Contact( #"AV-21.01".QCMD_OP )
   END_RUNG wire#w3
   // the same network as SCL:
   #"AV-21.01"(LOCK := #lock,   // "Valve"
               LIOP_SEL := #Init,
               L_AUT := #Init,
               L_REMOTE := #Init,
               L_RESET := #Reset,
               AUT_OP := "T-21.00_DB".QAV_Transfer,
               FB_OPEN := #"AV-21.01".QCMD_OP,
               FB_CLOSE := NOT #"AV-21.01".QCMD_OP,
               L_MON := #Init,
               INSTANCE := 'AV-21.01',
               QCMD_OP => "AV-21.01");
END_REGION

REGION Network 30: AV-21.02
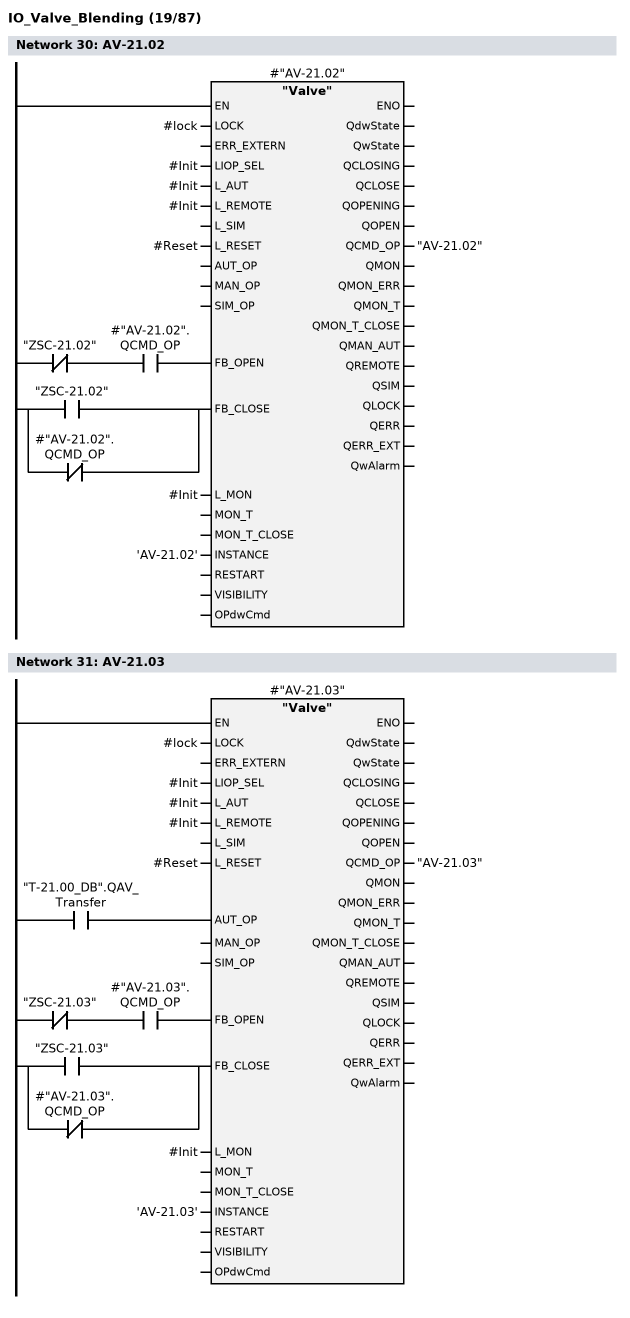
   RUNG wire#powerrail
      #"AV-21.02"(FB_OPEN := wire#w1, FB_CLOSE := wire#w2, LOCK := #lock, ERR_EXTERN :=, LIOP_SEL := #Init, L_AUT := #Init, L_REMOTE := #Init, L_SIM :=, L_RESET := #Reset, AUT_OP :=, MAN_OP :=, SIM_OP :=, L_MON := #Init, MON_T :=, MON_T_CLOSE :=, INSTANCE := 'AV-21.02', RESTART :=, VISIBILITY :=, OPdwCmd :=, QdwState =>, QwState =>, QCLOSING =>, QCLOSE =>, QOPENING =>, QOPEN =>, QCMD_OP => "AV-21.02", QMON =>, QMON_ERR =>, QMON_T =>, QMON_T_CLOSE =>, QMAN_AUT =>, QREMOTE =>, QSIM =>, QLOCK =>, QERR =>, QERR_EXT =>, QwAlarm =>)
   END_RUNG
   RUNG wire#powerrail
      I_Contact( "ZSC-21.02" )
      Contact( #"AV-21.02".QCMD_OP )
   END_RUNG wire#w1
   RUNG wire#powerrail
      Contact( "ZSC-21.02" )
   END_RUNG wire#w2
   RUNG wire#powerrail
      I_Contact( #"AV-21.02".QCMD_OP )
   END_RUNG wire#w2
   // the same network as SCL:
   #"AV-21.02"(LOCK := #lock,   // "Valve"
               LIOP_SEL := #Init,
               L_AUT := #Init,
               L_REMOTE := #Init,
               L_RESET := #Reset,
               FB_OPEN := NOT "ZSC-21.02" AND #"AV-21.02".QCMD_OP,
               FB_CLOSE := "ZSC-21.02" OR NOT #"AV-21.02".QCMD_OP,
               L_MON := #Init,
               INSTANCE := 'AV-21.02',
               QCMD_OP => "AV-21.02");
END_REGION

REGION Network 31: AV-21.03
   RUNG wire#powerrail
      #"AV-21.03"(AUT_OP := wire#w1, FB_OPEN := wire#w2, FB_CLOSE := wire#w3, LOCK := #lock, ERR_EXTERN :=, LIOP_SEL := #Init, L_AUT := #Init, L_REMOTE := #Init, L_SIM :=, L_RESET := #Reset, MAN_OP :=, SIM_OP :=, L_MON := #Init, MON_T :=, MON_T_CLOSE :=, INSTANCE := 'AV-21.03', RESTART :=, VISIBILITY :=, OPdwCmd :=, QdwState =>, QwState =>, QCLOSING =>, QCLOSE =>, QOPENING =>, QOPEN =>, QCMD_OP => "AV-21.03", QMON =>, QMON_ERR =>, QMON_T =>, QMON_T_CLOSE =>, QMAN_AUT =>, QREMOTE =>, QSIM =>, QLOCK =>, QERR =>, QERR_EXT =>, QwAlarm =>)
   END_RUNG
   RUNG wire#powerrail
      Contact( "T-21.00_DB".QAV_Transfer )
   END_RUNG wire#w1
   RUNG wire#powerrail
      I_Contact( "ZSC-21.03" )
      Contact( #"AV-21.03".QCMD_OP )
   END_RUNG wire#w2
   RUNG wire#powerrail
      Contact( "ZSC-21.03" )
   END_RUNG wire#w3
   RUNG wire#powerrail
      I_Contact( #"AV-21.03".QCMD_OP )
   END_RUNG wire#w3
   // the same network as SCL:
   #"AV-21.03"(LOCK := #lock,   // "Valve"
               LIOP_SEL := #Init,
               L_AUT := #Init,
               L_REMOTE := #Init,
               L_RESET := #Reset,
               AUT_OP := "T-21.00_DB".QAV_Transfer,
               FB_OPEN := NOT "ZSC-21.03" AND #"AV-21.03".QCMD_OP,
               FB_CLOSE := "ZSC-21.03" OR NOT #"AV-21.03".QCMD_OP,
               L_MON := #Init,
               INSTANCE := 'AV-21.03',
               QCMD_OP => "AV-21.03");
END_REGION

REGION Network 32: AV-21.04
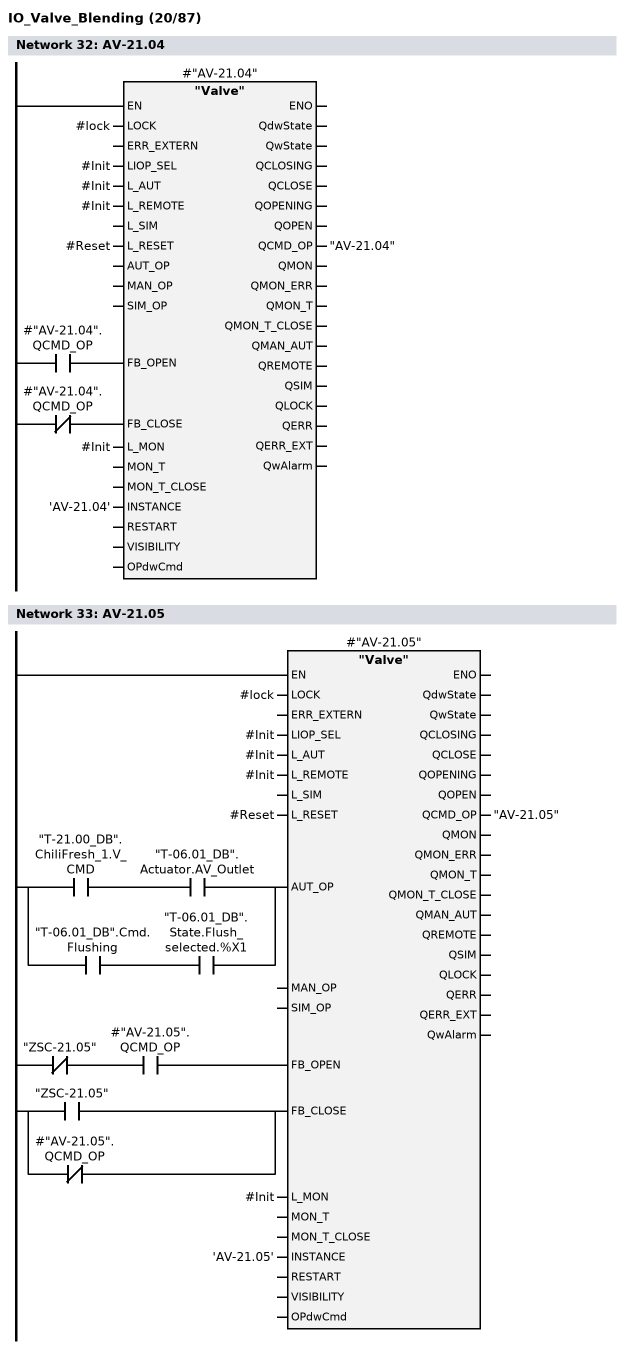
   RUNG wire#powerrail
      #"AV-21.04"(FB_OPEN := wire#w1, FB_CLOSE := wire#w2, LOCK := #lock, ERR_EXTERN :=, LIOP_SEL := #Init, L_AUT := #Init, L_REMOTE := #Init, L_SIM :=, L_RESET := #Reset, AUT_OP :=, MAN_OP :=, SIM_OP :=, L_MON := #Init, MON_T :=, MON_T_CLOSE :=, INSTANCE := 'AV-21.04', RESTART :=, VISIBILITY :=, OPdwCmd :=, QdwState =>, QwState =>, QCLOSING =>, QCLOSE =>, QOPENING =>, QOPEN =>, QCMD_OP => "AV-21.04", QMON =>, QMON_ERR =>, QMON_T =>, QMON_T_CLOSE =>, QMAN_AUT =>, QREMOTE =>, QSIM =>, QLOCK =>, QERR =>, QERR_EXT =>, QwAlarm =>)
   END_RUNG
   RUNG wire#powerrail
      Contact( #"AV-21.04".QCMD_OP )
   END_RUNG wire#w1
   RUNG wire#powerrail
      I_Contact( #"AV-21.04".QCMD_OP )
   END_RUNG wire#w2
   // the same network as SCL:
   #"AV-21.04"(LOCK := #lock,   // "Valve"
               LIOP_SEL := #Init,
               L_AUT := #Init,
               L_REMOTE := #Init,
               L_RESET := #Reset,
               FB_OPEN := #"AV-21.04".QCMD_OP,
               FB_CLOSE := NOT #"AV-21.04".QCMD_OP,
               L_MON := #Init,
               INSTANCE := 'AV-21.04',
               QCMD_OP => "AV-21.04");
END_REGION

REGION Network 33: AV-21.05
   RUNG wire#powerrail
      #"AV-21.05"(AUT_OP := wire#w1, FB_OPEN := wire#w2, FB_CLOSE := wire#w3, LOCK := #lock, ERR_EXTERN :=, LIOP_SEL := #Init, L_AUT := #Init, L_REMOTE := #Init, L_SIM :=, L_RESET := #Reset, MAN_OP :=, SIM_OP :=, L_MON := #Init, MON_T :=, MON_T_CLOSE :=, INSTANCE := 'AV-21.05', RESTART :=, VISIBILITY :=, OPdwCmd :=, QdwState =>, QwState =>, QCLOSING =>, QCLOSE =>, QOPENING =>, QOPEN =>, QCMD_OP => "AV-21.05", QMON =>, QMON_ERR =>, QMON_T =>, QMON_T_CLOSE =>, QMAN_AUT =>, QREMOTE =>, QSIM =>, QLOCK =>, QERR =>, QERR_EXT =>, QwAlarm =>)
   END_RUNG
   RUNG wire#powerrail
      Contact( "T-21.00_DB".ChiliFresh_1.V_CMD )
      Contact( "T-06.01_DB".Actuator.AV_Outlet )
   END_RUNG wire#w1
   RUNG wire#powerrail
      Contact( "T-06.01_DB".Cmd.Flushing )
      Contact( "T-06.01_DB".State.Flush_selected.%X1 )
   END_RUNG wire#w1
   RUNG wire#powerrail
      I_Contact( "ZSC-21.05" )
      Contact( #"AV-21.05".QCMD_OP )
   END_RUNG wire#w2
   RUNG wire#powerrail
      Contact( "ZSC-21.05" )
   END_RUNG wire#w3
   RUNG wire#powerrail
      I_Contact( #"AV-21.05".QCMD_OP )
   END_RUNG wire#w3
   // the same network as SCL:
   #"AV-21.05"(LOCK := #lock,   // "Valve"
               LIOP_SEL := #Init,
               L_AUT := #Init,
               L_REMOTE := #Init,
               L_RESET := #Reset,
               AUT_OP := ("T-21.00_DB".ChiliFresh_1.V_CMD AND "T-06.01_DB".Actuator.AV_Outlet) OR ("T-06.01_DB".Cmd.Flushing AND "T-06.01_DB".State.Flush_selected.%X1),
               FB_OPEN := NOT "ZSC-21.05" AND #"AV-21.05".QCMD_OP,
               FB_CLOSE := "ZSC-21.05" OR NOT #"AV-21.05".QCMD_OP,
               L_MON := #Init,
               INSTANCE := 'AV-21.05',
               QCMD_OP => "AV-21.05");
END_REGION

REGION Network 34: AV-21.06
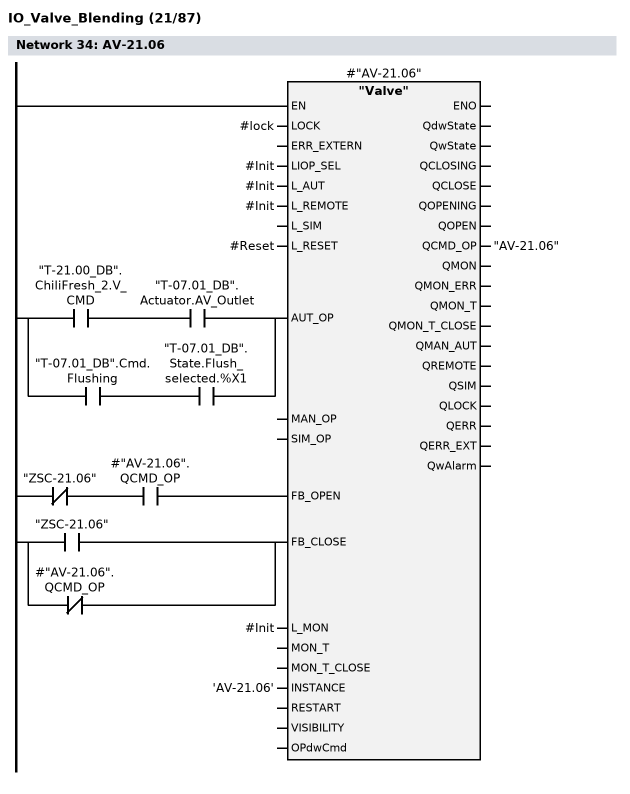
   RUNG wire#powerrail
      #"AV-21.06"(AUT_OP := wire#w1, FB_OPEN := wire#w2, FB_CLOSE := wire#w3, LOCK := #lock, ERR_EXTERN :=, LIOP_SEL := #Init, L_AUT := #Init, L_REMOTE := #Init, L_SIM :=, L_RESET := #Reset, MAN_OP :=, SIM_OP :=, L_MON := #Init, MON_T :=, MON_T_CLOSE :=, INSTANCE := 'AV-21.06', RESTART :=, VISIBILITY :=, OPdwCmd :=, QdwState =>, QwState =>, QCLOSING =>, QCLOSE =>, QOPENING =>, QOPEN =>, QCMD_OP => "AV-21.06", QMON =>, QMON_ERR =>, QMON_T =>, QMON_T_CLOSE =>, QMAN_AUT =>, QREMOTE =>, QSIM =>, QLOCK =>, QERR =>, QERR_EXT =>, QwAlarm =>)
   END_RUNG
   RUNG wire#powerrail
      Contact( "T-21.00_DB".ChiliFresh_2.V_CMD )
      Contact( "T-07.01_DB".Actuator.AV_Outlet )
   END_RUNG wire#w1
   RUNG wire#powerrail
      Contact( "T-07.01_DB".Cmd.Flushing )
      Contact( "T-07.01_DB".State.Flush_selected.%X1 )
   END_RUNG wire#w1
   RUNG wire#powerrail
      I_Contact( "ZSC-21.06" )
      Contact( #"AV-21.06".QCMD_OP )
   END_RUNG wire#w2
   RUNG wire#powerrail
      Contact( "ZSC-21.06" )
   END_RUNG wire#w3
   RUNG wire#powerrail
      I_Contact( #"AV-21.06".QCMD_OP )
   END_RUNG wire#w3
   // the same network as SCL:
   #"AV-21.06"(LOCK := #lock,   // "Valve"
               LIOP_SEL := #Init,
               L_AUT := #Init,
               L_REMOTE := #Init,
               L_RESET := #Reset,
               AUT_OP := ("T-21.00_DB".ChiliFresh_2.V_CMD AND "T-07.01_DB".Actuator.AV_Outlet) OR ("T-07.01_DB".Cmd.Flushing AND "T-07.01_DB".State.Flush_selected.%X1),
               FB_OPEN := NOT "ZSC-21.06" AND #"AV-21.06".QCMD_OP,
               FB_CLOSE := "ZSC-21.06" OR NOT #"AV-21.06".QCMD_OP,
               L_MON := #Init,
               INSTANCE := 'AV-21.06',
               QCMD_OP => "AV-21.06");
END_REGION

REGION Network 35: AV-21.07
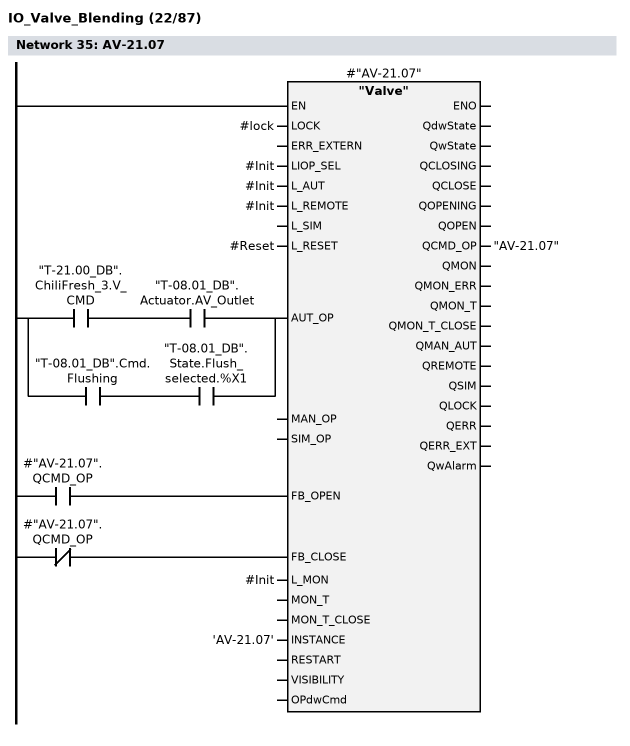
   RUNG wire#powerrail
      #"AV-21.07"(AUT_OP := wire#w1, FB_OPEN := wire#w2, FB_CLOSE := wire#w3, LOCK := #lock, ERR_EXTERN :=, LIOP_SEL := #Init, L_AUT := #Init, L_REMOTE := #Init, L_SIM :=, L_RESET := #Reset, MAN_OP :=, SIM_OP :=, L_MON := #Init, MON_T :=, MON_T_CLOSE :=, INSTANCE := 'AV-21.07', RESTART :=, VISIBILITY :=, OPdwCmd :=, QdwState =>, QwState =>, QCLOSING =>, QCLOSE =>, QOPENING =>, QOPEN =>, QCMD_OP => "AV-21.07", QMON =>, QMON_ERR =>, QMON_T =>, QMON_T_CLOSE =>, QMAN_AUT =>, QREMOTE =>, QSIM =>, QLOCK =>, QERR =>, QERR_EXT =>, QwAlarm =>)
   END_RUNG
   RUNG wire#powerrail
      Contact( "T-21.00_DB".ChiliFresh_3.V_CMD )
      Contact( "T-08.01_DB".Actuator.AV_Outlet )
   END_RUNG wire#w1
   RUNG wire#powerrail
      Contact( "T-08.01_DB".Cmd.Flushing )
      Contact( "T-08.01_DB".State.Flush_selected.%X1 )
   END_RUNG wire#w1
   RUNG wire#powerrail
      Contact( #"AV-21.07".QCMD_OP )
   END_RUNG wire#w2
   RUNG wire#powerrail
      I_Contact( #"AV-21.07".QCMD_OP )
   END_RUNG wire#w3
   // the same network as SCL:
   #"AV-21.07"(LOCK := #lock,   // "Valve"
               LIOP_SEL := #Init,
               L_AUT := #Init,
               L_REMOTE := #Init,
               L_RESET := #Reset,
               AUT_OP := ("T-21.00_DB".ChiliFresh_3.V_CMD AND "T-08.01_DB".Actuator.AV_Outlet) OR ("T-08.01_DB".Cmd.Flushing AND "T-08.01_DB".State.Flush_selected.%X1),
               FB_OPEN := #"AV-21.07".QCMD_OP,
               FB_CLOSE := NOT #"AV-21.07".QCMD_OP,
               L_MON := #Init,
               INSTANCE := 'AV-21.07',
               QCMD_OP => "AV-21.07");
END_REGION

REGION Network 36: AV-21.08
